LIN {X 0,Y 160.233,Z 340.194,A -85,B 0,C 180,E1 -26280.001,E2 -26280.001} C_VEL
LIN {X 0,Y 166.329,Z 331.475,A -85,B 0,C 180,E1 -26281.824,E2 -26281.824} C_VEL
LIN {X 0,Y 172.518,Z 320.915,A -85,B 0,C 180,E1 -26283.53,E2 -26283.53} C_VEL
LIN {X 0,Y 177.938,Z 309.578,A -85,B 0,C 180,E1 -26284.913,E2 -26284.913} C_VEL
LIN {X 0,Y 182.273,Z 298.101,A -85,B 0,C 180,E1 -26285.975,E2 -26285.975} C_VEL
LIN {X 0,Y 185.919,Z 285.028,A -85,B 0,C 180,E1 -26286.826,E2 -26286.826} C_VEL
LIN {X 0,Y 188.418,Z 271.569,A -85,B 0,C 180,E1 -26287.371,E2 -26287.371} C_VEL
LIN {X 0,Y 188.786,Z 268.726,A -85,B 0,C 180,E1 -26287.476,E2 -26287.476} C_VEL
LIN {X 0,Y 187.979,Z 266.198,A -85,B 0,C 180,E1 -26288.985,E2 -26288.985} C_VEL
LIN {X 0,Y 186.573,Z 263.076,A -85,B 0,C 180,E1 -26292.26,E2 -26292.26} C_VEL
LIN {X 0,Y 185.638,Z 260.546,A -85,B 0,C 180,E1 -26296.638,E2 -26296.638} C_VEL
LIN {X 0,Y 185.466,Z 260.699,A -85,B 0,C 180,E1 -26299.226,E2 -26299.226} C_VEL
LIN {X 0,Y 185.624,Z 261.538,A -85,B 0,C 180,E1 -26301.451,E2 -26301.451} C_VEL
LIN {X 0,Y 186.516,Z 265.492,A -85,B 0,C 180,E1 -26305.669,E2 -26305.669} C_VEL
LIN {X 0,Y 187.489,Z 269.73,A -85,B 0,C 180,E1 -26308.373,E2 -26308.373} C_VEL
LIN {X 0,Y 188.311,Z 273.021,A -85,B 0,C 180,E1 -26310.049,E2 -26310.049} C_VEL
LIN {X 0,Y 185.957,Z 286.979,A -85,B 0,C 180,E1 -26310.584,E2 -26310.584} C_VEL
LIN {X 0,Y 182.286,Z 300.423,A -85,B 0,C 180,E1 -26311.258,E2 -26311.258} C_VEL
LIN {X 0,Y 177.515,Z 313.155,A -85,B 0,C 180,E1 -26312.191,E2 -26312.191} C_VEL
LIN {X 0,Y 171.61,Z 325.353,A -85,B 0,C 180,E1 -26313.441,E2 -26313.441} C_VEL
LIN {X 0,Y 165.133,Z 336.315,A -85,B 0,C 180,E1 -26314.986,E2 -26314.986} C_VEL
LIN {X 0,Y 158.089,Z 346.198,A -85,B 0,C 180,E1 -26316.848,E2 -26316.848} C_VEL
LIN {X 0,Y 150.033,Z 355.815,A -85,B 0,C 180,E1 -26319.382,E2 -26319.382} C_VEL
LIN {X 0,Y 143.561,Z 362.421,A -85,B 0,C 180,E1 -26321.704,E2 -26321.704} C_VEL
LIN {X 0,Y 137.635,Z 367.953,A -85,B 0,C 180,E1 -26324.365,E2 -26324.365} C_VEL
LIN {X 0,Y 130.825,Z 373.459,A -85,B 0,C 180,E1 -26327.814,E2 -26327.814} C_VEL
LIN {X 0,Y 124.739,Z 377.873,A -85,B 0,C 180,E1 -26331.699,E2 -26331.699} C_VEL
LIN {X 0,Y 117.665,Z 382.218,A -85,B 0,C 180,E1 -26337.48,E2 -26337.48} C_VEL
LIN {X 0,Y 114.58,Z 383.794,A -85,B 0,C 180,E1 -26340.611,E2 -26340.611} C_VEL
LIN {X 0,Y 109.675,Z 385.745,A -85,B 0,C 180,E1 -26347.386,E2 -26347.386} C_VEL
LIN {X 0,Y 106.621,Z 386.253,A -85,B 0,C 180,E1 -26354.71,E2 -26354.71} C_VEL
LIN {X 0,Y 105.796,Z 385.958,A -85,B 0,C 180,E1 -26358.502,E2 -26358.502} C_VEL
LIN {X 0,Y 105.382,Z 384.173,A -85,B 0,C 180,E1 -26366.174,E2 -26366.174} C_VEL
LIN {X 0,Y 105.627,Z 382.684,A -85,B 0,C 180,E1 -26369.998,E2 -26369.998} C_VEL
LIN {X 0,Y 105.445,Z 379.479,A -85,B 0,C 180,E1 -26375.736,E2 -26375.736} C_VEL
LIN {X 0,Y 105.949,Z 375.143,A -85,B 0,C 180,E1 -26381.476,E2 -26381.476} C_VEL
LIN {X 0,Y 107.231,Z 369.534,A -85,B 0,C 180,E1 -26387.151,E2 -26387.151} C_VEL
LIN {X 0,Y 109.528,Z 362.495,A -85,B 0,C 180,E1 -26392.641,E2 -26392.641} C_VEL
LIN {X 0,Y 112.586,Z 353.593,A -85,B 0,C 180,E1 -26397.914,E2 -26397.914} C_VEL
LIN {X 0,Y 116.234,Z 343.804,A -85,B 0,C 180,E1 -26402.31,E2 -26402.31} C_VEL
LIN {X 0,Y 119.878,Z 333.229,A -85,B 0,C 180,E1 -26405.89,E2 -26405.89} C_VEL
LIN {X 0,Y 123.364,Z 321.863,A -85,B 0,C 180,E1 -26408.802,E2 -26408.802} C_VEL
LIN {X 0,Y 126.427,Z 310.142,A -85,B 0,C 180,E1 -26411.043,E2 -26411.043} C_VEL
LIN {X 0,Y 127.768,Z 304.244,A -85,B 0,C 180,E1 -26411.915,E2 -26411.915} C_VEL
LIN {X 0,Y 128.3,Z 298.694,A -85,B 0,C 180,E1 -26412.766,E2 -26412.766} C_VEL
LIN {X 0,Y 127.436,Z 289.443,A -85,B 0,C 180,E1 -26414.362,E2 -26414.362} C_VEL
LIN {X 0,Y 126.129,Z 280.088,A -85,B 0,C 180,E1 -26415.771,E2 -26415.771} C_VEL
LIN {X 0,Y 126.029,Z 274.273,A -85,B 0,C 180,E1 -26416.291,E2 -26416.291} C_VEL
LIN {X 0,Y 128.319,Z 245.916,A -85,B 0,C 180,E1 -26417.859,E2 -26417.859} C_VEL
LIN {X 0,Y 127.617,Z 235.927,A -85,B 0,C 180,E1 -26418.895,E2 -26418.895} C_VEL
LIN {X 0,Y 122.358,Z 220.14,A -85,B 0,C 180,E1 -26422.064,E2 -26422.064} C_VEL
LIN {X 0,Y 116.899,Z 206.665,A -85,B 0,C 180,E1 -26425.56,E2 -26425.56} C_VEL
LIN {X 0,Y 111.473,Z 197.493,A -85,B 0,C 180,E1 -26429.052,E2 -26429.052} C_VEL
LIN {X 0,Y 108.315,Z 192.741,A -85,B 0,C 180,E1 -26431.276,E2 -26431.276} C_VEL
LIN {X 0,Y 106.676,Z 190.164,A -85,B 0,C 180,E1 -26432.535,E2 -26432.535} C_VEL
LIN {X 0,Y 104.643,Z 187.418,A -85,B 0,C 180,E1 -26434.114,E2 -26434.114} C_VEL
LIN {X 0,Y 103.842,Z 185.904,A -85,B 0,C 180,E1 -26434.814,E2 -26434.814} C_VEL
LIN {X 0,Y 101.804,Z 183.712,A -85,B 0,C 180,E1 -26436.475,E2 -26436.475} C_VEL
LIN {X 0,Y 100.819,Z 180.918,A -85,B 0,C 180,E1 -26437.723,E2 -26437.723} C_VEL
LIN {X 0,Y 101.094,Z 180.891,A -85,B 0,C 180,E1 -26446.713,E2 -26446.713} C_VEL
LIN {X 0,Y 101.261,Z 180.849,A -85,B 0,C 180,E1 -26452.019,E2 -26452.019} C_VEL
LIN {X 0,Y 101.867,Z 180.78,A -85,B 0,C 180,E1 -26459.998,E2 -26459.998} C_VEL
LIN {X 0,Y 101.264,Z 180.871,A -85,B 0,C 180,E1 -26467.976,E2 -26467.976} C_VEL
LIN {X 0,Y 101.121,Z 180.858,A -85,B 0,C 180,E1 -26473.351,E2 -26473.351} C_VEL
LIN {X 0,Y 100.815,Z 180.924,A -85,B 0,C 180,E1 -26480.397,E2 -26480.397} C_VEL
LIN {X 0,Y 100.77,Z 180.899,A -85,B 0,C 180,E1 -26484.957,E2 -26484.957} C_VEL
LIN {X 0,Y 100.706,Z 180.927,A -85,B 0,C 180,E1 -26493.133,E2 -26493.133} C_VEL
LIN {X 0,Y 100.723,Z 180.929,A -85,B 0,C 180,E1 -26499.871,E2 -26499.871} C_VEL
LIN {X 0,Y 100.749,Z 180.912,A -85,B 0,C 180,E1 -26505.77,E2 -26505.77} C_VEL
LIN {X 0,Y 100.727,Z 180.937,A -85,B 0,C 180,E1 -26511.103,E2 -26511.103} C_VEL
LIN {X 0,Y 100.707,Z 180.933,A -85,B 0,C 180,E1 -26516.866,E2 -26516.866} C_VEL
LIN {X 0,Y 100.677,Z 180.943,A -85,B 0,C 180,E1 -26521.175,E2 -26521.175} C_VEL
LIN {X 0,Y 101.611,Z 183.625,A -85,B 0,C 180,E1 -26522.235,E2 -26522.235} C_VEL
LIN {X 0,Y 103.67,Z 185.856,A -85,B 0,C 180,E1 -26523.923,E2 -26523.923} C_VEL
LIN {X 0,Y 104.397,Z 186.604,A -85,B 0,C 180,E1 -26524.484,E2 -26524.484} C_VEL
LIN {X 0,Y 106.409,Z 189.752,A -85,B 0,C 180,E1 -26526.107,E2 -26526.107} C_VEL
LIN {X 0,Y 107.849,Z 191.69,A -85,B 0,C 180,E1 -26527.194,E2 -26527.194} C_VEL
LIN {X 0,Y 112.897,Z 199.282,A -85,B 0,C 180,E1 -26530.72,E2 -26530.72} C_VEL
LIN {X 0,Y 117.907,Z 207.42,A -85,B 0,C 180,E1 -26533.807,E2 -26533.807} C_VEL
LIN {X 0,Y 125.125,Z 221.433,A -85,B 0,C 180,E1 -26537.922,E2 -26537.922} C_VEL
LIN {X 0,Y 129.197,Z 232.015,A -85,B 0,C 180,E1 -26540.167,E2 -26540.167} C_VEL
LIN {X 0,Y 125.432,Z 274.357,A -85,B 0,C 180,E1 -26542.51,E2 -26542.51} C_VEL
LIN {X 0,Y 123.412,Z 288.198,A -85,B 0,C 180,E1 -26543.872,E2 -26543.872} C_VEL
LIN {X 0,Y 121.046,Z 300.183,A -85,B 0,C 180,E1 -26545.632,E2 -26545.632} C_VEL
LIN {X 0,Y 117.924,Z 312.467,A -85,B 0,C 180,E1 -26548.124,E2 -26548.124} C_VEL
LIN {X 0,Y 114.128,Z 324.389,A -85,B 0,C 180,E1 -26551.325,E2 -26551.325} C_VEL
LIN {X 0,Y 110.537,Z 334.612,A -85,B 0,C 180,E1 -26555.018,E2 -26555.018} C_VEL
LIN {X 0,Y 106.892,Z 344.199,A -85,B 0,C 180,E1 -26559.534,E2 -26559.534} C_VEL
LIN {X 0,Y 103.736,Z 352.637,A -85,B 0,C 180,E1 -26564.72,E2 -26564.72} C_VEL
LIN {X 0,Y 101.152,Z 359.661,A -85,B 0,C 180,E1 -26570.331,E2 -26570.331} C_VEL
LIN {X 0,Y 99.286,Z 365.396,A -85,B 0,C 180,E1 -26576.26,E2 -26576.26} C_VEL
LIN {X 0,Y 98.025,Z 370.249,A -85,B 0,C 180,E1 -26582.849,E2 -26582.849} C_VEL
LIN {X 0,Y 97.822,Z 374.211,A -85,B 0,C 180,E1 -26590.289,E2 -26590.289} C_VEL
LIN {X 0,Y 98.496,Z 376.154,A -85,B 0,C 180,E1 -26595.526,E2 -26595.526} C_VEL
LIN {X 0,Y 99.918,Z 377.48,A -85,B 0,C 180,E1 -26600.728,E2 -26600.728} C_VEL
LIN {X 0,Y 102.418,Z 378.187,A -85,B 0,C 180,E1 -26606.707,E2 -26606.707} C_VEL
LIN {X 0,Y 105.825,Z 378.009,A -85,B 0,C 180,E1 -26612.3,E2 -26612.3} C_VEL
LIN {X 0,Y 110.113,Z 376.968,A -85,B 0,C 180,E1 -26617.486,E2 -26617.486} C_VEL
LIN {X 0,Y 117.115,Z 374.207,A -85,B 0,C 180,E1 -26623.778,E2 -26623.778} C_VEL
LIN {X 0,Y 124.851,Z 370.01,A -85,B 0,C 180,E1 -26629.013,E2 -26629.013} C_VEL
LIN {X 0,Y 132.704,Z 364.735,A -85,B 0,C 180,E1 -26633.233,E2 -26633.233} C_VEL
LIN {X 0,Y 140.792,Z 358.262,A -85,B 0,C 180,E1 -26636.742,E2 -26636.742} C_VEL
LIN {X 0,Y 148.978,Z 350.375,A -85,B 0,C 180,E1 -26639.778,E2 -26639.778} C_VEL
LIN {X 0,Y 157.176,Z 341.077,A -85,B 0,C 180,E1 -26642.302,E2 -26642.302} C_VEL
LIN {X 0,Y 164.233,Z 331.414,A -85,B 0,C 180,E1 -26644.264,E2 -26644.264} C_VEL
LIN {X 0,Y 170.344,Z 321.314,A -85,B 0,C 180,E1 -26645.802,E2 -26645.802} C_VEL
LIN {X 0,Y 176.076,Z 309.663,A -85,B 0,C 180,E1 -26647.155,E2 -26647.155} C_VEL
LIN {X 0,Y 180.601,Z 297.942,A -85,B 0,C 180,E1 -26648.173,E2 -26648.173} C_VEL
LIN {X 0,Y 184.166,Z 285.441,A -85,B 0,C 180,E1 -26648.946,E2 -26648.946} C_VEL
LIN {X 0,Y 186.585,Z 273.08,A -85,B 0,C 180,E1 -26649.439,E2 -26649.439} C_VEL
LIN {X 0,Y 185.37,Z 269.984,A -85,B 0,C 180,E1 -26652.607,E2 -26652.607} C_VEL
LIN {X 0,Y 184.57,Z 267.581,A -85,B 0,C 180,E1 -26656.737,E2 -26656.737} C_VEL
LIN {X 0,Y 184.407,Z 267.621,A -85,B 0,C 180,E1 -26658.78,E2 -26658.78} C_VEL
LIN {X 0,Y 184.513,Z 268.464,A -85,B 0,C 180,E1 -26661.046,E2 -26661.046} C_VEL
LIN {X 0,Y 185.168,Z 272.044,A -85,B 0,C 180,E1 -26664.925,E2 -26664.925} C_VEL
LIN {X 0,Y 185.924,Z 276.177,A -85,B 0,C 180,E1 -26667.586,E2 -26667.586} C_VEL
LIN {X 0,Y 186.077,Z 277.273,A -85,B 0,C 180,E1 -26668.108,E2 -26668.108} C_VEL
LIN {X 0,Y 183.263,Z 290.946,A -85,B 0,C 180,E1 -26668.62,E2 -26668.62} C_VEL
LIN {X 0,Y 179.064,Z 304.295,A -85,B 0,C 180,E1 -26669.333,E2 -26669.333} C_VEL
LIN {X 0,Y 173.92,Z 316.593,A -85,B 0,C 180,E1 -26670.257,E2 -26670.257} C_VEL
LIN {X 0,Y 167.904,Z 327.975,A -85,B 0,C 180,E1 -26671.475,E2 -26671.475} C_VEL
LIN {X 0,Y 160.499,Z 339.366,A -85,B 0,C 180,E1 -26673.125,E2 -26673.125} C_VEL
LIN {X 0,Y 154.007,Z 347.754,A -85,B 0,C 180,E1 -26674.77,E2 -26674.77} C_VEL
LIN {X 0,Y 145.684,Z 356.975,A -85,B 0,C 180,E1 -26677.249,E2 -26677.249} C_VEL
LIN {X 0,Y 138.98,Z 363.363,A -85,B 0,C 180,E1 -26679.538,E2 -26679.538} C_VEL
LIN {X 0,Y 132.809,Z 368.671,A -85,B 0,C 180,E1 -26682.193,E2 -26682.193} C_VEL
LIN {X 0,Y 125.673,Z 373.97,A -85,B 0,C 180,E1 -26685.648,E2 -26685.648} C_VEL
LIN {X 0,Y 119.246,Z 378.166,A -85,B 0,C 180,E1 -26689.583,E2 -26689.583} C_VEL
LIN {X 0,Y 111.733,Z 382.295,A -85,B 0,C 180,E1 -26695.519,E2 -26695.519} C_VEL
LIN {X 0,Y 105.609,Z 384.82,A -85,B 0,C 180,E1 -26702.233,E2 -26702.233} C_VEL
LIN {X 0,Y 101.151,Z 385.886,A -85,B 0,C 180,E1 -26709.669,E2 -26709.669} C_VEL
LIN {X 0,Y 98.835,Z 385.455,A -85,B 0,C 180,E1 -26717.68,E2 -26717.68} C_VEL
LIN {X 0,Y 98.306,Z 383.517,A -85,B 0,C 180,E1 -26725.898,E2 -26725.898} C_VEL
LIN {X 0,Y 98.573,Z 381.956,A -85,B 0,C 180,E1 -26729.998,E2 -26729.998} C_VEL
LIN {X 0,Y 98.39,Z 378.59,A -85,B 0,C 180,E1 -26736.148,E2 -26736.148} C_VEL
LIN {X 0,Y 98.984,Z 374.082,A -85,B 0,C 180,E1 -26742.296,E2 -26742.296} C_VEL
LIN {X 0,Y 100.799,Z 367.149,A -85,B 0,C 180,E1 -26749.338,E2 -26749.338} C_VEL
LIN {X 0,Y 103.505,Z 359.608,A -85,B 0,C 180,E1 -26755.109,E2 -26755.109} C_VEL
LIN {X 0,Y 106.341,Z 351.85,A -85,B 0,C 180,E1 -26759.711,E2 -26759.711} C_VEL
LIN {X 0,Y 110.101,Z 342.13,A -85,B 0,C 180,E1 -26764.115,E2 -26764.115} C_VEL
LIN {X 0,Y 113.71,Z 332.002,A -85,B 0,C 180,E1 -26767.612,E2 -26767.612} C_VEL
LIN {X 0,Y 117.42,Z 320.485,A -85,B 0,C 180,E1 -26770.608,E2 -26770.608} C_VEL
LIN {X 0,Y 120.653,Z 308.395,A -85,B 0,C 180,E1 -26772.903,E2 -26772.903} C_VEL
LIN {X 0,Y 123.371,Z 295.237,A -85,B 0,C 180,E1 -26774.68,E2 -26774.68} C_VEL
LIN {X 0,Y 125.293,Z 282.442,A -85,B 0,C 180,E1 -26775.799,E2 -26775.799} C_VEL
LIN {X 0,Y 126.029,Z 274.273,A -85,B 0,C 180,E1 -26776.291,E2 -26776.291} C_VEL
LIN {X 0,Y 126.035,Z 268.462,A -85,B 0,C 180,E1 -26776.759,E2 -26776.759} C_VEL
LIN {X 0,Y 124.727,Z 259.017,A -85,B 0,C 180,E1 -26777.932,E2 -26777.932} C_VEL
LIN {X 0,Y 123.318,Z 251.52,A -85,B 0,C 180,E1 -26779.016,E2 -26779.016} C_VEL
LIN {X 0,Y 122.351,Z 243.901,A -85,B 0,C 180,E1 -26779.997,E2 -26779.997} C_VEL
LIN {X 0,Y 121.929,Z 238.108,A -85,B 0,C 180,E1 -26780.649,E2 -26780.649} C_VEL
LIN {X 0,Y 117.441,Z 224.046,A -85,B 0,C 180,E1 -26783.657,E2 -26783.657} C_VEL
LIN {X 0,Y 112.403,Z 211.152,A -85,B 0,C 180,E1 -26787.163,E2 -26787.163} C_VEL
LIN {X 0,Y 107.107,Z 201.943,A -85,B 0,C 180,E1 -26790.905,E2 -26790.905} C_VEL
LIN {X 0,Y 102.944,Z 195.483,A -85,B 0,C 180,E1 -26794.212,E2 -26794.212} C_VEL
LIN {X 0,Y 100.08,Z 191.295,A -85,B 0,C 180,E1 -26796.694,E2 -26796.694} C_VEL
LIN {X 0,Y 97.932,Z 188.228,A -85,B 0,C 180,E1 -26798.73,E2 -26798.73} C_VEL
LIN {X 0,Y 97.319,Z 187.092,A -85,B 0,C 180,E1 -26799.385,E2 -26799.385} C_VEL
LIN {X 0,Y 95.008,Z 185.052,A -85,B 0,C 180,E1 -26801.674,E2 -26801.674} C_VEL
LIN {X 0,Y 93.897,Z 182.427,A -85,B 0,C 180,E1 -26803.132,E2 -26803.132} C_VEL
LIN {X 0,Y 93.809,Z 181.783,A -85,B 0,C 180,E1 -26803.394,E2 -26803.394} C_VEL
LIN {X 0,Y 94.062,Z 181.768,A -85,B 0,C 180,E1 -26807.045,E2 -26807.045} C_VEL
LIN {X 0,Y 94.192,Z 181.73,A -85,B 0,C 180,E1 -26811.416,E2 -26811.416} C_VEL
LIN {X 0,Y 94.793,Z 181.659,A -85,B 0,C 180,E1 -26819.998,E2 -26819.998} C_VEL
LIN {X 0,Y 94.197,Z 181.751,A -85,B 0,C 180,E1 -26828.579,E2 -26828.579} C_VEL
LIN {X 0,Y 94.039,Z 181.739,A -85,B 0,C 180,E1 -26833.708,E2 -26833.708} C_VEL
LIN {X 0,Y 93.69,Z 181.802,A -85,B 0,C 180,E1 -26842.026,E2 -26842.026} C_VEL
LIN {X 0,Y 93.619,Z 181.791,A -85,B 0,C 180,E1 -26846.768,E2 -26846.768} C_VEL
LIN {X 0,Y 93.618,Z 181.799,A -85,B 0,C 180,E1 -26854.336,E2 -26854.336} C_VEL
LIN {X 0,Y 93.645,Z 181.814,A -85,B 0,C 180,E1 -26862.486,E2 -26862.486} C_VEL
LIN {X 0,Y 93.644,Z 181.808,A -85,B 0,C 180,E1 -26868.63,E2 -26868.63} C_VEL
LIN {X 0,Y 93.605,Z 181.809,A -85,B 0,C 180,E1 -26875.354,E2 -26875.354} C_VEL
LIN {X 0,Y 94.576,Z 184.497,A -85,B 0,C 180,E1 -26876.699,E2 -26876.699} C_VEL
LIN {X 0,Y 96.422,Z 186.628,A -85,B 0,C 180,E1 -26878.655,E2 -26878.655} C_VEL
LIN {X 0,Y 97.443,Z 187.526,A -85,B 0,C 180,E1 -26879.636,E2 -26879.636} C_VEL
LIN {X 0,Y 99.279,Z 190.545,A -85,B 0,C 180,E1 -26881.492,E2 -26881.492} C_VEL
LIN {X 0,Y 101.113,Z 192.633,A -85,B 0,C 180,E1 -26883.086,E2 -26883.086} C_VEL
LIN {X 0,Y 104.658,Z 197.834,A -85,B 0,C 180,E1 -26886.016,E2 -26886.016} C_VEL
LIN {X 0,Y 109.424,Z 205.272,A -85,B 0,C 180,E1 -26889.593,E2 -26889.593} C_VEL
LIN {X 0,Y 113.895,Z 212.833,A -85,B 0,C 180,E1 -26892.573,E2 -26892.573} C_VEL
LIN {X 0,Y 120.275,Z 225.658,A -85,B 0,C 180,E1 -26896.485,E2 -26896.485} C_VEL
LIN {X 0,Y 123.282,Z 234.132,A -85,B 0,C 180,E1 -26898.353,E2 -26898.353} C_VEL
LIN {X 0,Y 119.557,Z 274.458,A -85,B 0,C 180,E1 -26900.646,E2 -26900.646} C_VEL
LIN {X 0,Y 117.566,Z 287.596,A -85,B 0,C 180,E1 -26901.948,E2 -26901.948} C_VEL
LIN {X 0,Y 115.013,Z 300.17,A -85,B 0,C 180,E1 -26903.82,E2 -26903.82} C_VEL
LIN {X 0,Y 111.733,Z 312.533,A -85,B 0,C 180,E1 -26906.396,E2 -26906.396} C_VEL
LIN {X 0,Y 107.971,Z 323.898,A -85,B 0,C 180,E1 -26909.536,E2 -26909.536} C_VEL
LIN {X 0,Y 104.172,Z 334.203,A -85,B 0,C 180,E1 -26913.328,E2 -26913.328} C_VEL
LIN {X 0,Y 100.316,Z 343.88,A -85,B 0,C 180,E1 -26918.057,E2 -26918.057} C_VEL
LIN {X 0,Y 96.901,Z 352.544,A -85,B 0,C 180,E1 -26923.636,E2 -26923.636} C_VEL
LIN {X 0,Y 94.146,Z 359.676,A -85,B 0,C 180,E1 -26929.631,E2 -26929.631} C_VEL
LIN {X 0,Y 92.247,Z 365.25,A -85,B 0,C 180,E1 -26935.712,E2 -26935.712} C_VEL
LIN {X 0,Y 90.942,Z 370.167,A -85,B 0,C 180,E1 -26942.752,E2 -26942.752} C_VEL
LIN {X 0,Y 90.663,Z 373.561,A -85,B 0,C 180,E1 -26949.183,E2 -26949.183} C_VEL
LIN {X 0,Y 91.501,Z 376.25,A -85,B 0,C 180,E1 -26956.272,E2 -26956.272} C_VEL
LIN {X 0,Y 93.466,Z 377.886,A -85,B 0,C 180,E1 -26963.022,E2 -26963.022} C_VEL
LIN {X 0,Y 97.027,Z 378.582,A -85,B 0,C 180,E1 -26970.371,E2 -26970.371} C_VEL
LIN {X 0,Y 100.488,Z 378.319,A -85,B 0,C 180,E1 -26975.402,E2 -26975.402} C_VEL
LIN {X 0,Y 105.082,Z 377.273,A -85,B 0,C 180,E1 -26980.466,E2 -26980.466} C_VEL
LIN {X 0,Y 110.669,Z 375.334,A -85,B 0,C 180,E1 -26985.287,E2 -26985.287} C_VEL
LIN {X 0,Y 118.62,Z 371.612,A -85,B 0,C 180,E1 -26990.613,E2 -26990.613} C_VEL
LIN {X 0,Y 126.986,Z 366.619,A -85,B 0,C 180,E1 -26995.028,E2 -26995.028} C_VEL
LIN {X 0,Y 136.401,Z 359.72,A -85,B 0,C 180,E1 -26998.966,E2 -26998.966} C_VEL
LIN {X 0,Y 144.141,Z 352.917,A -85,B 0,C 180,E1 -27001.695,E2 -27001.695} C_VEL
LIN {X 0,Y 152.381,Z 344.374,A -85,B 0,C 180,E1 -27004.134,E2 -27004.134} C_VEL
LIN {X 0,Y 159.988,Z 334.827,A -85,B 0,C 180,E1 -27006.145,E2 -27006.145} C_VEL
LIN {X 0,Y 167.299,Z 323.756,A -85,B 0,C 180,E1 -27007.875,E2 -27007.875} C_VEL
LIN {X 0,Y 173.592,Z 311.856,A -85,B 0,C 180,E1 -27009.254,E2 -27009.254} C_VEL
LIN {X 0,Y 178.572,Z 299.834,A -85,B 0,C 180,E1 -27010.283,E2 -27010.283} C_VEL
LIN {X 0,Y 182.504,Z 287.095,A -85,B 0,C 180,E1 -27011.064,E2 -27011.064} C_VEL
LIN {X 0,Y 184.447,Z 278.319,A -85,B 0,C 180,E1 -27011.452,E2 -27011.452} C_VEL
LIN {X 0,Y 183.966,Z 276.707,A -85,B 0,C 180,E1 -27013.252,E2 -27013.252} C_VEL
LIN {X 0,Y 183.408,Z 274.517,A -85,B 0,C 180,E1 -27017.349,E2 -27017.349} C_VEL
LIN {X 0,Y 183.365,Z 275.226,A -85,B 0,C 180,E1 -27020.466,E2 -27020.466} C_VEL
LIN {X 0,Y 183.767,Z 278.831,A -85,B 0,C 180,E1 -27024.334,E2 -27024.334} C_VEL
LIN {X 0,Y 184.052,Z 281.28,A -85,B 0,C 180,E1 -27026.017,E2 -27026.017} C_VEL
LIN {X 0,Y 180.937,Z 294.125,A -85,B 0,C 180,E1 -27026.571,E2 -27026.571} C_VEL
LIN {X 0,Y 176.384,Z 307.158,A -85,B 0,C 180,E1 -27027.274,E2 -27027.274} C_VEL
LIN {X 0,Y 170.542,Z 319.74,A -85,B 0,C 180,E1 -27028.251,E2 -27028.251} C_VEL
LIN {X 0,Y 163.604,Z 331.66,A -85,B 0,C 180,E1 -27029.552,E2 -27029.552} C_VEL
LIN {X 0,Y 156.042,Z 342.234,A -85,B 0,C 180,E1 -27031.155,E2 -27031.155} C_VEL
LIN {X 0,Y 148.685,Z 350.91,A -85,B 0,C 180,E1 -27032.962,E2 -27032.962} C_VEL
LIN {X 0,Y 140.143,Z 359.482,A -85,B 0,C 180,E1 -27035.418,E2 -27035.418} C_VEL
LIN {X 0,Y 133.38,Z 365.329,A -85,B 0,C 180,E1 -27037.777,E2 -27037.777} C_VEL
LIN {X 0,Y 125.63,Z 371.178,A -85,B 0,C 180,E1 -27040.953,E2 -27040.953} C_VEL
LIN {X 0,Y 118.362,Z 375.9,A -85,B 0,C 180,E1 -27044.556,E2 -27044.556} C_VEL
LIN {X 0,Y 111.826,Z 379.58,A -85,B 0,C 180,E1 -27048.705,E2 -27048.705} C_VEL
LIN {X 0,Y 105.949,Z 382.339,A -85,B 0,C 180,E1 -27053.342,E2 -27053.342} C_VEL
LIN {X 0,Y 99.35,Z 384.688,A -85,B 0,C 180,E1 -27060.316,E2 -27060.316} C_VEL
LIN {X 0,Y 94.499,Z 385.54,A -85,B 0,C 180,E1 -27068.167,E2 -27068.167} C_VEL
LIN {X 0,Y 91.905,Z 384.931,A -85,B 0,C 180,E1 -27076.735,E2 -27076.735} C_VEL
LIN {X 0,Y 91.255,Z 382.854,A -85,B 0,C 180,E1 -27085.58,E2 -27085.58} C_VEL
LIN {X 0,Y 91.498,Z 381.166,A -85,B 0,C 180,E1 -27089.997,E2 -27089.997} C_VEL
LIN {X 0,Y 91.36,Z 377.649,A -85,B 0,C 180,E1 -27096.624,E2 -27096.624} C_VEL
LIN {X 0,Y 92.028,Z 372.948,A -85,B 0,C 180,E1 -27103.242,E2 -27103.242} C_VEL
LIN {X 0,Y 93.705,Z 366.932,A -85,B 0,C 180,E1 -27109.722,E2 -27109.722} C_VEL
LIN {X 0,Y 96.535,Z 359.419,A -85,B 0,C 180,E1 -27115.898,E2 -27115.898} C_VEL
LIN {X 0,Y 99.513,Z 351.69,A -85,B 0,C 180,E1 -27120.796,E2 -27120.796} C_VEL
LIN {X 0,Y 103.226,Z 342.6,A -85,B 0,C 180,E1 -27125.21,E2 -27125.21} C_VEL
LIN {X 0,Y 107.237,Z 331.939,A -85,B 0,C 180,E1 -27129.106,E2 -27129.106} C_VEL
LIN {X 0,Y 111.095,Z 320.47,A -85,B 0,C 180,E1 -27132.231,E2 -27132.231} C_VEL
LIN {X 0,Y 114.459,Z 308.497,A -85,B 0,C 180,E1 -27134.608,E2 -27134.608} C_VEL
LIN {X 0,Y 117.417,Z 294.939,A -85,B 0,C 180,E1 -27136.495,E2 -27136.495} C_VEL
LIN {X 0,Y 119.428,Z 281.907,A -85,B 0,C 180,E1 -27137.665,E2 -27137.665} C_VEL
LIN {X 0,Y 122.51,Z 246.783,A -85,B 0,C 180,E1 -27139.693,E2 -27139.693} C_VEL
LIN {X 0,Y 122.351,Z 243.901,A -85,B 0,C 180,E1 -27139.997,E2 -27139.997} C_VEL
LIN {X 0,Y 121.71,Z 240.236,A -85,B 0,C 180,E1 -27140.543,E2 -27140.543} C_VEL
LIN {X 0,Y 120.468,Z 236.88,A -85,B 0,C 180,E1 -27141.295,E2 -27141.295} C_VEL
LIN {X 0,Y 116.944,Z 230.966,A -85,B 0,C 180,E1 -27143.21,E2 -27143.21} C_VEL
LIN {X 0,Y 111.045,Z 222.501,A -85,B 0,C 180,E1 -27146.641,E2 -27146.641} C_VEL
LIN {X 0,Y 109.458,Z 219.349,A -85,B 0,C 180,E1 -27147.733,E2 -27147.733} C_VEL
LIN {X 0,Y 107.063,Z 213.848,A -85,B 0,C 180,E1 -27149.574,E2 -27149.574} C_VEL
LIN {X 0,Y 101.847,Z 204.644,A -85,B 0,C 180,E1 -27153.77,E2 -27153.77} C_VEL
LIN {X 0,Y 98.777,Z 200.068,A -85,B 0,C 180,E1 -27156.435,E2 -27156.435} C_VEL
LIN {X 0,Y 96.5,Z 196.602,A -85,B 0,C 180,E1 -27158.643,E2 -27158.643} C_VEL
LIN {X 0,Y 94.108,Z 193.001,A -85,B 0,C 180,E1 -27161.21,E2 -27161.21} C_VEL
LIN {X 0,Y 91.854,Z 190.437,A -85,B 0,C 180,E1 -27163.752,E2 -27163.752} C_VEL
LIN {X 0,Y 90.636,Z 188.067,A -85,B 0,C 180,E1 -27165.401,E2 -27165.401} C_VEL
LIN {X 0,Y 88.164,Z 185.728,A -85,B 0,C 180,E1 -27168.648,E2 -27168.648} C_VEL
LIN {X 0,Y 87.181,Z 183.289,A -85,B 0,C 180,E1 -27170.427,E2 -27170.427} C_VEL
LIN {X 0,Y 87.107,Z 182.614,A -85,B 0,C 180,E1 -27170.858,E2 -27170.858} C_VEL
LIN {X 0,Y 87.72,Z 182.539,A -85,B 0,C 180,E1 -27179.997,E2 -27179.997} C_VEL
LIN {X 0,Y 87.105,Z 182.631,A -85,B 0,C 180,E1 -27189.284,E2 -27189.284} C_VEL
LIN {X 0,Y 86.946,Z 182.622,A -85,B 0,C 180,E1 -27194.085,E2 -27194.085} C_VEL
LIN {X 0,Y 86.66,Z 182.687,A -85,B 0,C 180,E1 -27198.926,E2 -27198.926} C_VEL
LIN {X 0,Y 86.581,Z 182.667,A -85,B 0,C 180,E1 -27206.766,E2 -27206.766} C_VEL
LIN {X 0,Y 86.546,Z 182.672,A -85,B 0,C 180,E1 -27215.707,E2 -27215.707} C_VEL
LIN {X 0,Y 86.569,Z 182.69,A -85,B 0,C 180,E1 -27223.063,E2 -27223.063} C_VEL
LIN {X 0,Y 86.63,Z 182.783,A -85,B 0,C 180,E1 -27227.559,E2 -27227.559} C_VEL
LIN {X 0,Y 87.432,Z 185.323,A -85,B 0,C 180,E1 -27229.204,E2 -27229.204} C_VEL
LIN {X 0,Y 89.292,Z 187.497,A -85,B 0,C 180,E1 -27231.909,E2 -27231.909} C_VEL
LIN {X 0,Y 90.834,Z 188.586,A -85,B 0,C 180,E1 -27233.786,E2 -27233.786} C_VEL
LIN {X 0,Y 92.752,Z 191.879,A -85,B 0,C 180,E1 -27236.231,E2 -27236.231} C_VEL
LIN {X 0,Y 94.494,Z 193.623,A -85,B 0,C 180,E1 -27238.077,E2 -27238.077} C_VEL
LIN {X 0,Y 96.836,Z 197.115,A -85,B 0,C 180,E1 -27240.56,E2 -27240.56} C_VEL
LIN {X 0,Y 98.225,Z 199.073,A -85,B 0,C 180,E1 -27241.898,E2 -27241.898} C_VEL
LIN {X 0,Y 101.072,Z 203.296,A -85,B 0,C 180,E1 -27244.444,E2 -27244.444} C_VEL
LIN {X 0,Y 107.252,Z 213.206,A -85,B 0,C 180,E1 -27249.314,E2 -27249.314} C_VEL
LIN {X 0,Y 112.021,Z 222.621,A -85,B 0,C 180,E1 -27252.7,E2 -27252.7} C_VEL
LIN {X 0,Y 115.461,Z 229.809,A -85,B 0,C 180,E1 -27254.908,E2 -27254.908} C_VEL
LIN {X 0,Y 117.569,Z 235.73,A -85,B 0,C 180,E1 -27256.337,E2 -27256.337} C_VEL
LIN {X 0,Y 113.833,Z 274.465,A -85,B 0,C 180,E1 -27258.583,E2 -27258.583} C_VEL
LIN {X 0,Y 111.733,Z 287.778,A -85,B 0,C 180,E1 -27259.927,E2 -27259.927} C_VEL
LIN {X 0,Y 109.004,Z 300.609,A -85,B 0,C 180,E1 -27261.894,E2 -27261.894} C_VEL
LIN {X 0,Y 105.678,Z 312.537,A -85,B 0,C 180,E1 -27264.452,E2 -27264.452} C_VEL
LIN {X 0,Y 101.928,Z 323.393,A -85,B 0,C 180,E1 -27267.532,E2 -27267.532} C_VEL
LIN {X 0,Y 97.941,Z 333.704,A -85,B 0,C 180,E1 -27271.425,E2 -27271.425} C_VEL
LIN {X 0,Y 93.759,Z 343.649,A -85,B 0,C 180,E1 -27276.458,E2 -27276.458} C_VEL
LIN {X 0,Y 90.101,Z 352.388,A -85,B 0,C 180,E1 -27282.389,E2 -27282.389} C_VEL
LIN {X 0,Y 87.176,Z 359.594,A -85,B 0,C 180,E1 -27288.815,E2 -27288.815} C_VEL
LIN {X 0,Y 85.256,Z 364.899,A -85,B 0,C 180,E1 -27294.944,E2 -27294.944} C_VEL
LIN {X 0,Y 83.803,Z 370.256,A -85,B 0,C 180,E1 -27303.009,E2 -27303.009} C_VEL
LIN {X 0,Y 83.768,Z 374.566,A -85,B 0,C 180,E1 -27312.163,E2 -27312.163} C_VEL
LIN {X 0,Y 84.821,Z 376.692,A -85,B 0,C 180,E1 -27318.486,E2 -27318.486} C_VEL
LIN {X 0,Y 87.186,Z 378.281,A -85,B 0,C 180,E1 -27325.652,E2 -27325.652} C_VEL
LIN {X 0,Y 90.621,Z 378.929,A -85,B 0,C 180,E1 -27332.272,E2 -27332.272} C_VEL
LIN {X 0,Y 96.973,Z 378.366,A -85,B 0,C 180,E1 -27340.425,E2 -27340.425} C_VEL
LIN {X 0,Y 101.852,Z 377.194,A -85,B 0,C 180,E1 -27345.032,E2 -27345.032} C_VEL
LIN {X 0,Y 110.274,Z 374.09,A -85,B 0,C 180,E1 -27351.074,E2 -27351.074} C_VEL
LIN {X 0,Y 119.739,Z 369.398,A -85,B 0,C 180,E1 -27356.229,E2 -27356.229} C_VEL
LIN {X 0,Y 128.707,Z 363.752,A -85,B 0,C 180,E1 -27360.002,E2 -27360.002} C_VEL
LIN {X 0,Y 136.958,Z 357.466,A -85,B 0,C 180,E1 -27362.943,E2 -27362.943} C_VEL
LIN {X 0,Y 145.64,Z 349.596,A -85,B 0,C 180,E1 -27365.54,E2 -27365.54} C_VEL
LIN {X 0,Y 153.843,Z 340.752,A -85,B 0,C 180,E1 -27367.628,E2 -27367.628} C_VEL
LIN {X 0,Y 161.133,Z 331.247,A -85,B 0,C 180,E1 -27369.305,E2 -27369.305} C_VEL
LIN {X 0,Y 168.118,Z 320.188,A -85,B 0,C 180,E1 -27370.759,E2 -27370.759} C_VEL
LIN {X 0,Y 173.05,Z 310.61,A -85,B 0,C 180,E1 -27371.717,E2 -27371.717} C_VEL
LIN {X 0,Y 178.017,Z 298.517,A -85,B 0,C 180,E1 -27372.648,E2 -27372.648} C_VEL
LIN {X 0,Y 181.661,Z 286.463,A -85,B 0,C 180,E1 -27373.314,E2 -27373.314} C_VEL
LIN {X 0,Y 182.368,Z 283.593,A -85,B 0,C 180,E1 -27373.441,E2 -27373.441} C_VEL
LIN {X 0,Y 182.04,Z 281.453,A -85,B 0,C 180,E1 -27377.483,E2 -27377.483} C_VEL
LIN {X 0,Y 181.958,Z 282.19,A -85,B 0,C 180,E1 -27380.18,E2 -27380.18} C_VEL
LIN {X 0,Y 182.026,Z 285.356,A -85,B 0,C 180,E1 -27383.633,E2 -27383.633} C_VEL
LIN {X 0,Y 181.981,Z 286.157,A -85,B 0,C 180,E1 -27384.04,E2 -27384.04} C_VEL
LIN {X 0,Y 177.8,Z 300.258,A -85,B 0,C 180,E1 -27384.611,E2 -27384.611} C_VEL
LIN {X 0,Y 172.667,Z 312.695,A -85,B 0,C 180,E1 -27385.339,E2 -27385.339} C_VEL
LIN {X 0,Y 166.581,Z 324.252,A -85,B 0,C 180,E1 -27386.291,E2 -27386.291} C_VEL
LIN {X 0,Y 159.525,Z 335.164,A -85,B 0,C 180,E1 -27387.545,E2 -27387.545} C_VEL
LIN {X 0,Y 151.025,Z 345.842,A -85,B 0,C 180,E1 -27389.242,E2 -27389.242} C_VEL
LIN {X 0,Y 142.041,Z 355.276,A -85,B 0,C 180,E1 -27391.401,E2 -27391.401} C_VEL
LIN {X 0,Y 133.309,Z 362.957,A -85,B 0,C 180,E1 -27393.864,E2 -27393.864} C_VEL
LIN {X 0,Y 126.48,Z 368.203,A -85,B 0,C 180,E1 -27396.318,E2 -27396.318} C_VEL
LIN {X 0,Y 118.5,Z 373.429,A -85,B 0,C 180,E1 -27399.553,E2 -27399.553} C_VEL
LIN {X 0,Y 111.129,Z 377.563,A -85,B 0,C 180,E1 -27403.338,E2 -27403.338} C_VEL
LIN {X 0,Y 103.95,Z 380.96,A -85,B 0,C 180,E1 -27408.051,E2 -27408.051} C_VEL
LIN {X 0,Y 96.565,Z 383.66,A -85,B 0,C 180,E1 -27414.389,E2 -27414.389} C_VEL
LIN {X 0,Y 90.328,Z 385.026,A -85,B 0,C 180,E1 -27422.168,E2 -27422.168} C_VEL
LIN {X 0,Y 86.166,Z 384.967,A -85,B 0,C 180,E1 -27430.955,E2 -27430.955} C_VEL
LIN {X 0,Y 84.319,Z 383.454,A -85,B 0,C 180,E1 -27440.401,E2 -27440.401} C_VEL
LIN {X 0,Y 84.371,Z 380.975,A -85,B 0,C 180,E1 -27448.439,E2 -27448.439} C_VEL
LIN {X 0,Y 84.371,Z 379.654,A -85,B 0,C 180,E1 -27451.55,E2 -27451.55} C_VEL
LIN {X 0,Y 84.489,Z 375.177,A -85,B 0,C 180,E1 -27459.574,E2 -27459.574} C_VEL
LIN {X 0,Y 85.931,Z 368.855,A -85,B 0,C 180,E1 -27467.858,E2 -27467.858} C_VEL
LIN {X 0,Y 88.485,Z 361.935,A -85,B 0,C 180,E1 -27474.641,E2 -27474.641} C_VEL
LIN {X 0,Y 91.358,Z 354.799,A -85,B 0,C 180,E1 -27479.999,E2 -27479.999} C_VEL
LIN {X 0,Y 95.074,Z 346.184,A -85,B 0,C 180,E1 -27484.949,E2 -27484.949} C_VEL
LIN {X 0,Y 99.481,Z 335.588,A -85,B 0,C 180,E1 -27489.478,E2 -27489.478} C_VEL
LIN {X 0,Y 103.316,Z 325.068,A -85,B 0,C 180,E1 -27492.859,E2 -27492.859} C_VEL
LIN {X 0,Y 106.997,Z 313.524,A -85,B 0,C 180,E1 -27495.584,E2 -27495.584} C_VEL
LIN {X 0,Y 110.346,Z 300.509,A -85,B 0,C 180,E1 -27497.763,E2 -27497.763} C_VEL
LIN {X 0,Y 112.89,Z 287.206,A -85,B 0,C 180,E1 -27499.259,E2 -27499.259} C_VEL
LIN {X 0,Y 114.63,Z 271.795,A -85,B 0,C 180,E1 -27500.312,E2 -27500.312} C_VEL
LIN {X 0,Y 116.828,Z 246.797,A -85,B 0,C 180,E1 -27501.78,E2 -27501.78} C_VEL
LIN {X 0,Y 116.412,Z 240.265,A -85,B 0,C 180,E1 -27502.555,E2 -27502.555} C_VEL
LIN {X 0,Y 112.025,Z 226.294,A -85,B 0,C 180,E1 -27505.8,E2 -27505.8} C_VEL
LIN {X 0,Y 109.458,Z 219.349,A -85,B 0,C 180,E1 -27507.733,E2 -27507.733} C_VEL
LIN {X 0,Y 107.022,Z 215.1,A -85,B 0,C 180,E1 -27509.464,E2 -27509.464} C_VEL
LIN {X 0,Y 104.026,Z 211.727,A -85,B 0,C 180,E1 -27511.559,E2 -27511.559} C_VEL
LIN {X 0,Y 93.599,Z 202.612,A -85,B 0,C 180,E1 -27520.135,E2 -27520.135} C_VEL
LIN {X 0,Y 91.05,Z 198.848,A -85,B 0,C 180,E1 -27523.1,E2 -27523.1} C_VEL
LIN {X 0,Y 88.584,Z 195.488,A -85,B 0,C 180,E1 -27526.228,E2 -27526.228} C_VEL
LIN {X 0,Y 87.886,Z 194.192,A -85,B 0,C 180,E1 -27527.27,E2 -27527.27} C_VEL
LIN {X 0,Y 85.437,Z 191.268,A -85,B 0,C 180,E1 -27531.012,E2 -27531.012} C_VEL
LIN {X 0,Y 84.663,Z 189.302,A -85,B 0,C 180,E1 -27532.605,E2 -27532.605} C_VEL
LIN {X 0,Y 82.175,Z 187.433,A -85,B 0,C 180,E1 -27537.24,E2 -27537.24} C_VEL
LIN {X 0,Y 80.31,Z 183.452,A -85,B 0,C 180,E1 -27542.819,E2 -27542.819} C_VEL
LIN {X 0,Y 79.99,Z 183.508,A -85,B 0,C 180,E1 -27550.118,E2 -27550.118} C_VEL
LIN {X 0,Y 79.762,Z 183.519,A -85,B 0,C 180,E1 -27555.325,E2 -27555.325} C_VEL
LIN {X 0,Y 79.519,Z 183.575,A -85,B 0,C 180,E1 -27560.7,E2 -27560.7} C_VEL
LIN {X 0,Y 79.48,Z 183.556,A -85,B 0,C 180,E1 -27567.847,E2 -27567.847} C_VEL
LIN {X 0,Y 79.498,Z 183.692,A -85,B 0,C 180,E1 -27573.918,E2 -27573.918} C_VEL
LIN {X 0,Y 80.58,Z 186.632,A -85,B 0,C 180,E1 -27578.045,E2 -27578.045} C_VEL
LIN {X 0,Y 83.667,Z 189.183,A -85,B 0,C 180,E1 -27584.704,E2 -27584.704} C_VEL
LIN {X 0,Y 84.374,Z 189.721,A -85,B 0,C 180,E1 -27585.921,E2 -27585.921} C_VEL
LIN {X 0,Y 85.823,Z 192.606,A -85,B 0,C 180,E1 -27588.673,E2 -27588.673} C_VEL
LIN {X 0,Y 88.241,Z 194.979,A -85,B 0,C 180,E1 -27592.169,E2 -27592.169} C_VEL
LIN {X 0,Y 90.598,Z 198.538,A -85,B 0,C 180,E1 -27595.307,E2 -27595.307} C_VEL
LIN {X 0,Y 91.783,Z 200.057,A -85,B 0,C 180,E1 -27596.687,E2 -27596.687} C_VEL
LIN {X 0,Y 95.205,Z 205.053,A -85,B 0,C 180,E1 -27600.43,E2 -27600.43} C_VEL
LIN {X 0,Y 99.259,Z 211.459,A -85,B 0,C 180,E1 -27604.298,E2 -27604.298} C_VEL
LIN {X 0,Y 104.406,Z 220.417,A -85,B 0,C 180,E1 -27608.556,E2 -27608.556} C_VEL
LIN {X 0,Y 110.509,Z 233.459,A -85,B 0,C 180,E1 -27613.109,E2 -27613.109} C_VEL
LIN {X 0,Y 111.915,Z 237.552,A -85,B 0,C 180,E1 -27614.153,E2 -27614.153} C_VEL
LIN {X 0,Y 108.275,Z 274.095,A -85,B 0,C 180,E1 -27616.321,E2 -27616.321} C_VEL
LIN {X 0,Y 106.052,Z 287.64,A -85,B 0,C 180,E1 -27617.691,E2 -27617.691} C_VEL
LIN {X 0,Y 103.187,Z 300.541,A -85,B 0,C 180,E1 -27619.703,E2 -27619.703} C_VEL
LIN {X 0,Y 99.55,Z 312.886,A -85,B 0,C 180,E1 -27622.417,E2 -27622.417} C_VEL
LIN {X 0,Y 95.416,Z 324.214,A -85,B 0,C 180,E1 -27625.778,E2 -27625.778} C_VEL
LIN {X 0,Y 91.134,Z 334.708,A -85,B 0,C 180,E1 -27630.003,E2 -27630.003} C_VEL
LIN {X 0,Y 87.286,Z 343.343,A -85,B 0,C 180,E1 -27634.621,E2 -27634.621} C_VEL
LIN {X 0,Y 83.379,Z 352.181,A -85,B 0,C 180,E1 -27640.935,E2 -27640.935} C_VEL
LIN {X 0,Y 79.983,Z 360.091,A -85,B 0,C 180,E1 -27648.503,E2 -27648.503} C_VEL
LIN {X 0,Y 77.631,Z 366.535,A -85,B 0,C 180,E1 -27656.917,E2 -27656.917} C_VEL
LIN {X 0,Y 76.574,Z 370.833,A -85,B 0,C 180,E1 -27664.312,E2 -27664.312} C_VEL
LIN {X 0,Y 76.72,Z 374.556,A -85,B 0,C 180,E1 -27672.879,E2 -27672.879} C_VEL
LIN {X 0,Y 78.954,Z 377.638,A -85,B 0,C 180,E1 -27683.243,E2 -27683.243} C_VEL
LIN {X 0,Y 81.538,Z 378.768,A -85,B 0,C 180,E1 -27689.54,E2 -27689.54} C_VEL
LIN {X 0,Y 85.083,Z 379.295,A -85,B 0,C 180,E1 -27695.609,E2 -27695.609} C_VEL
LIN {X 0,Y 90.102,Z 379.03,A -85,B 0,C 180,E1 -27701.823,E2 -27701.823} C_VEL
LIN {X 0,Y 96.005,Z 377.913,A -85,B 0,C 180,E1 -27707.316,E2 -27707.316} C_VEL
LIN {X 0,Y 102.728,Z 375.916,A -85,B 0,C 180,E1 -27712.138,E2 -27712.138} C_VEL
LIN {X 0,Y 112.552,Z 371.873,A -85,B 0,C 180,E1 -27717.581,E2 -27717.581} C_VEL
LIN {X 0,Y 121.202,Z 367.225,A -85,B 0,C 180,E1 -27721.292,E2 -27721.292} C_VEL
LIN {X 0,Y 130.433,Z 361.143,A -85,B 0,C 180,E1 -27724.547,E2 -27724.547} C_VEL
LIN {X 0,Y 139.987,Z 353.518,A -85,B 0,C 180,E1 -27727.359,E2 -27727.359} C_VEL
LIN {X 0,Y 148.137,Z 345.728,A -85,B 0,C 180,E1 -27729.327,E2 -27729.327} C_VEL
LIN {X 0,Y 156.461,Z 336.098,A -85,B 0,C 180,E1 -27731.15,E2 -27731.15} C_VEL
LIN {X 0,Y 163.768,Z 325.825,A -85,B 0,C 180,E1 -27732.582,E2 -27732.582} C_VEL
LIN {X 0,Y 170.581,Z 314.083,A -85,B 0,C 180,E1 -27733.802,E2 -27733.802} C_VEL
LIN {X 0,Y 175.775,Z 302.617,A -85,B 0,C 180,E1 -27734.705,E2 -27734.705} C_VEL
LIN {X 0,Y 180.249,Z 289.537,A -85,B 0,C 180,E1 -27735.433,E2 -27735.433} C_VEL
LIN {X 0,Y 180.313,Z 288.432,A -85,B 0,C 180,E1 -27737.331,E2 -27737.331} C_VEL
LIN {X 0,Y 180.211,Z 288.918,A -85,B 0,C 180,E1 -27739.685,E2 -27739.685} C_VEL
LIN {X 0,Y 180.013,Z 290.91,A -85,B 0,C 180,E1 -27741.963,E2 -27741.963} C_VEL
LIN {X 0,Y 175.622,Z 303.703,A -85,B 0,C 180,E1 -27742.489,E2 -27742.489} C_VEL
LIN {X 0,Y 170.128,Z 315.804,A -85,B 0,C 180,E1 -27743.197,E2 -27743.197} C_VEL
LIN {X 0,Y 163.629,Z 327.09,A -85,B 0,C 180,E1 -27744.114,E2 -27744.114} C_VEL
LIN {X 0,Y 155.635,Z 338.403,A -85,B 0,C 180,E1 -27745.422,E2 -27745.422} C_VEL
LIN {X 0,Y 147.743,Z 347.618,A -85,B 0,C 180,E1 -27746.881,E2 -27746.881} C_VEL
LIN {X 0,Y 138.521,Z 356.585,A -85,B 0,C 180,E1 -27748.928,E2 -27748.928} C_VEL
LIN {X 0,Y 128.052,Z 365.006,A -85,B 0,C 180,E1 -27751.708,E2 -27751.708} C_VEL
LIN {X 0,Y 119.621,Z 370.749,A -85,B 0,C 180,E1 -27754.658,E2 -27754.658} C_VEL
LIN {X 0,Y 111.485,Z 375.386,A -85,B 0,C 180,E1 -27757.997,E2 -27757.997} C_VEL
LIN {X 0,Y 103.949,Z 378.997,A -85,B 0,C 180,E1 -27761.948,E2 -27761.948} C_VEL
LIN {X 0,Y 94.902,Z 382.424,A -85,B 0,C 180,E1 -27768.199,E2 -27768.199} C_VEL
LIN {X 0,Y 87.244,Z 384.324,A -85,B 0,C 180,E1 -27775.671,E2 -27775.671} C_VEL
LIN {X 0,Y 81.44,Z 384.8,A -85,B 0,C 180,E1 -27784.435,E2 -27784.435} C_VEL
LIN {X 0,Y 78.101,Z 383.82,A -85,B 0,C 180,E1 -27794.335,E2 -27794.335} C_VEL
LIN {X 0,Y 77.15,Z 381.334,A -85,B 0,C 180,E1 -27804.77,E2 -27804.77} C_VEL
LIN {X 0,Y 77.4,Z 379.483,A -85,B 0,C 180,E1 -27809.997,E2 -27809.997} C_VEL
LIN {X 0,Y 77.3,Z 375.623,A -85,B 0,C 180,E1 -27817.835,E2 -27817.835} C_VEL
LIN {X 0,Y 78.528,Z 369.565,A -85,B 0,C 180,E1 -27826.907,E2 -27826.907} C_VEL
LIN {X 0,Y 80.991,Z 362.882,A -85,B 0,C 180,E1 -27834.339,E2 -27834.339} C_VEL
LIN {X 0,Y 84.557,Z 354.525,A -85,B 0,C 180,E1 -27841.294,E2 -27841.294} C_VEL
LIN {X 0,Y 88.47,Z 345.943,A -85,B 0,C 180,E1 -27846.566,E2 -27846.566} C_VEL
LIN {X 0,Y 93.111,Z 335.346,A -85,B 0,C 180,E1 -27851.355,E2 -27851.355} C_VEL
LIN {X 0,Y 97.148,Z 324.925,A -85,B 0,C 180,E1 -27854.854,E2 -27854.854} C_VEL
LIN {X 0,Y 101,Z 313.471,A -85,B 0,C 180,E1 -27857.671,E2 -27857.671} C_VEL
LIN {X 0,Y 104.505,Z 300.577,A -85,B 0,C 180,E1 -27859.901,E2 -27859.901} C_VEL
LIN {X 0,Y 107.067,Z 287.939,A -85,B 0,C 180,E1 -27861.399,E2 -27861.399} C_VEL
LIN {X 0,Y 108.699,Z 275.448,A -85,B 0,C 180,E1 -27862.326,E2 -27862.326} C_VEL
LIN {X 0,Y 111.316,Z 248.04,A -85,B 0,C 180,E1 -27863.942,E2 -27863.942} C_VEL
LIN {X 0,Y 111.048,Z 242.742,A -85,B 0,C 180,E1 -27864.584,E2 -27864.584} C_VEL
LIN {X 0,Y 107.15,Z 229.813,A -85,B 0,C 180,E1 -27867.764,E2 -27867.764} C_VEL
LIN {X 0,Y 103.3,Z 219.28,A -85,B 0,C 180,E1 -27871.069,E2 -27871.069} C_VEL
LIN {X 0,Y 98.182,Z 209.936,A -85,B 0,C 180,E1 -27875.515,E2 -27875.515} C_VEL
LIN {X 0,Y 93.599,Z 202.612,A -85,B 0,C 180,E1 -27880.135,E2 -27880.135} C_VEL
LIN {X 0,Y 90.917,Z 200.122,A -85,B 0,C 180,E1 -27883.01,E2 -27883.01} C_VEL
LIN {X 0,Y 86.32,Z 197.732,A -85,B 0,C 180,E1 -27888.465,E2 -27888.465} C_VEL
LIN {X 0,Y 81.675,Z 195.369,A -85,B 0,C 180,E1 -27895.864,E2 -27895.864} C_VEL
LIN {X 0,Y 80.504,Z 194.146,A -85,B 0,C 180,E1 -27898.423,E2 -27898.423} C_VEL
LIN {X 0,Y 78.823,Z 190.504,A -85,B 0,C 180,E1 -27903.831,E2 -27903.831} C_VEL
LIN {X 0,Y 76.387,Z 189.79,A -85,B 0,C 180,E1 -27916.019,E2 -27916.019} C_VEL
LIN {X 0,Y 77.978,Z 190.513,A -85,B 0,C 180,E1 -27932.349,E2 -27932.349} C_VEL
LIN {X 0,Y 79.066,Z 193.36,A -85,B 0,C 180,E1 -27936.876,E2 -27936.876} C_VEL
LIN {X 0,Y 82.234,Z 196.266,A -85,B 0,C 180,E1 -27944.241,E2 -27944.241} C_VEL
LIN {X 0,Y 83.993,Z 199.373,A -85,B 0,C 180,E1 -27947.671,E2 -27947.671} C_VEL
LIN {X 0,Y 85.929,Z 201.568,A -85,B 0,C 180,E1 -27950.749,E2 -27950.749} C_VEL
LIN {X 0,Y 89.169,Z 206.439,A -85,B 0,C 180,E1 -27955.273,E2 -27955.273} C_VEL
LIN {X 0,Y 92.011,Z 210.663,A -85,B 0,C 180,E1 -27958.599,E2 -27958.599} C_VEL
LIN {X 0,Y 95.676,Z 216.828,A -85,B 0,C 180,E1 -27962.5,E2 -27962.5} C_VEL
LIN {X 0,Y 100.15,Z 224.884,A -85,B 0,C 180,E1 -27966.582,E2 -27966.582} C_VEL
LIN {X 0,Y 105.79,Z 237.408,A -85,B 0,C 180,E1 -27971.235,E2 -27971.235} C_VEL
LIN {X 0,Y 106.467,Z 239.818,A -85,B 0,C 180,E1 -27971.841,E2 -27971.841} C_VEL
LIN {X 0,Y 102.646,Z 275.109,A -85,B 0,C 180,E1 -27973.933,E2 -27973.933} C_VEL
LIN {X 0,Y 100.263,Z 289.056,A -85,B 0,C 180,E1 -27975.443,E2 -27975.443} C_VEL
LIN {X 0,Y 97.25,Z 301.578,A -85,B 0,C 180,E1 -27977.481,E2 -27977.481} C_VEL
LIN {X 0,Y 93.418,Z 313.702,A -85,B 0,C 180,E1 -27980.257,E2 -27980.257} C_VEL
LIN {X 0,Y 89.03,Z 325.022,A -85,B 0,C 180,E1 -27983.771,E2 -27983.771} C_VEL
LIN {X 0,Y 84.365,Z 335.736,A -85,B 0,C 180,E1 -27988.385,E2 -27988.385} C_VEL
LIN {X 0,Y 80.051,Z 344.917,A -85,B 0,C 180,E1 -27993.778,E2 -27993.778} C_VEL
LIN {X 0,Y 75.914,Z 353.6,A -85,B 0,C 180,E1 -28000.673,E2 -28000.673} C_VEL
LIN {X 0,Y 72.737,Z 360.699,A -85,B 0,C 180,E1 -28008.305,E2 -28008.305} C_VEL
LIN {X 0,Y 70.263,Z 367.322,A -85,B 0,C 180,E1 -28018.032,E2 -28018.032} C_VEL
LIN {X 0,Y 69.396,Z 372.033,A -85,B 0,C 180,E1 -28027.424,E2 -28027.424} C_VEL
LIN {X 0,Y 70.435,Z 376.054,A -85,B 0,C 180,E1 -28038.481,E2 -28038.481} C_VEL
LIN {X 0,Y 73.782,Z 378.535,A -85,B 0,C 180,E1 -28049.02,E2 -28049.02} C_VEL
LIN {X 0,Y 77.235,Z 379.432,A -85,B 0,C 180,E1 -28055.506,E2 -28055.506} C_VEL
LIN {X 0,Y 81.545,Z 379.643,A -85,B 0,C 180,E1 -28061.458,E2 -28061.458} C_VEL
LIN {X 0,Y 86.641,Z 379.249,A -85,B 0,C 180,E1 -28066.767,E2 -28066.767} C_VEL
LIN {X 0,Y 92.397,Z 378.182,A -85,B 0,C 180,E1 -28071.442,E2 -28071.442} C_VEL
LIN {X 0,Y 102.145,Z 375.293,A -85,B 0,C 180,E1 -28077.475,E2 -28077.475} C_VEL
LIN {X 0,Y 112.542,Z 370.894,A -85,B 0,C 180,E1 -28082.29,E2 -28082.29} C_VEL
LIN {X 0,Y 122.235,Z 365.642,A -85,B 0,C 180,E1 -28085.733,E2 -28085.733} C_VEL
LIN {X 0,Y 131.471,Z 359.441,A -85,B 0,C 180,E1 -28088.515,E2 -28088.515} C_VEL
LIN {X 0,Y 141.291,Z 351.386,A -85,B 0,C 180,E1 -28090.925,E2 -28090.925} C_VEL
LIN {X 0,Y 150.465,Z 342.301,A -85,B 0,C 180,E1 -28092.82,E2 -28092.82} C_VEL
LIN {X 0,Y 158.747,Z 332.268,A -85,B 0,C 180,E1 -28094.361,E2 -28094.361} C_VEL
LIN {X 0,Y 166.443,Z 320.758,A -85,B 0,C 180,E1 -28095.641,E2 -28095.641} C_VEL
LIN {X 0,Y 172.748,Z 308.836,A -85,B 0,C 180,E1 -28096.631,E2 -28096.631} C_VEL
LIN {X 0,Y 177.894,Z 296.05,A -85,B 0,C 180,E1 -28097.403,E2 -28097.403} C_VEL
LIN {X 0,Y 178.192,Z 295.183,A -85,B 0,C 180,E1 -28097.544,E2 -28097.544} C_VEL
LIN {X 0,Y 178.123,Z 295.424,A -85,B 0,C 180,E1 -28099.085,E2 -28099.085} C_VEL
LIN {X 0,Y 178.021,Z 295.86,A -85,B 0,C 180,E1 -28099.609,E2 -28099.609} C_VEL
LIN {X 0,Y 177.395,Z 297.733,A -85,B 0,C 180,E1 -28099.93,E2 -28099.93} C_VEL
LIN {X 0,Y 172.528,Z 309.683,A -85,B 0,C 180,E1 -28100.456,E2 -28100.456} C_VEL
LIN {X 0,Y 166.709,Z 320.827,A -85,B 0,C 180,E1 -28101.132,E2 -28101.132} C_VEL
LIN {X 0,Y 159.304,Z 332.176,A -85,B 0,C 180,E1 -28102.107,E2 -28102.107} C_VEL
LIN {X 0,Y 151.154,Z 342.406,A -85,B 0,C 180,E1 -28103.318,E2 -28103.318} C_VEL
LIN {X 0,Y 143.127,Z 350.83,A -85,B 0,C 180,E1 -28104.71,E2 -28104.71} C_VEL
LIN {X 0,Y 133.722,Z 359.147,A -85,B 0,C 180,E1 -28106.684,E2 -28106.684} C_VEL
LIN {X 0,Y 124.5,Z 365.928,A -85,B 0,C 180,E1 -28108.954,E2 -28108.954} C_VEL
LIN {X 0,Y 115.756,Z 371.401,A -85,B 0,C 180,E1 -28111.785,E2 -28111.785} C_VEL
LIN {X 0,Y 107.277,Z 375.809,A -85,B 0,C 180,E1 -28115.021,E2 -28115.021} C_VEL
LIN {X 0,Y 99.34,Z 379.255,A -85,B 0,C 180,E1 -28118.899,E2 -28118.899} C_VEL
LIN {X 0,Y 89.724,Z 382.416,A -85,B 0,C 180,E1 -28125.17,E2 -28125.17} C_VEL
LIN {X 0,Y 81.457,Z 384.128,A -85,B 0,C 180,E1 -28132.843,E2 -28132.843} C_VEL
LIN {X 0,Y 75.077,Z 384.38,A -85,B 0,C 180,E1 -28142.089,E2 -28142.089} C_VEL
LIN {X 0,Y 71.279,Z 383.193,A -85,B 0,C 180,E1 -28152.791,E2 -28152.791} C_VEL
LIN {X 0,Y 70.121,Z 380.551,A -85,B 0,C 180,E1 -28164.244,E2 -28164.244} C_VEL
LIN {X 0,Y 70.289,Z 378.289,A -85,B 0,C 180,E1 -28170.682,E2 -28170.682} C_VEL
LIN {X 0,Y 70.272,Z 374.546,A -85,B 0,C 180,E1 -28178.625,E2 -28178.625} C_VEL
LIN {X 0,Y 71.761,Z 368.248,A -85,B 0,C 180,E1 -28188.556,E2 -28188.556} C_VEL
LIN {X 0,Y 74.547,Z 361.339,A -85,B 0,C 180,E1 -28196.6,E2 -28196.6} C_VEL
LIN {X 0,Y 77.8,Z 354.237,A -85,B 0,C 180,E1 -28202.817,E2 -28202.817} C_VEL
LIN {X 0,Y 81.955,Z 345.669,A -85,B 0,C 180,E1 -28208.438,E2 -28208.438} C_VEL
LIN {X 0,Y 86.827,Z 335.119,A -85,B 0,C 180,E1 -28213.466,E2 -28213.466} C_VEL
LIN {X 0,Y 91.113,Z 324.671,A -85,B 0,C 180,E1 -28217.116,E2 -28217.116} C_VEL
LIN {X 0,Y 95.158,Z 313.244,A -85,B 0,C 180,E1 -28220.015,E2 -28220.015} C_VEL
LIN {X 0,Y 98.826,Z 300.378,A -85,B 0,C 180,E1 -28222.29,E2 -28222.29} C_VEL
LIN {X 0,Y 101.675,Z 286.905,A -85,B 0,C 180,E1 -28223.884,E2 -28223.884} C_VEL
LIN {X 0,Y 103.496,Z 272.448,A -85,B 0,C 180,E1 -28224.931,E2 -28224.931} C_VEL
LIN {X 0,Y 105.884,Z 248.49,A -85,B 0,C 180,E1 -28226.369,E2 -28226.369} C_VEL
LIN {X 0,Y 105.675,Z 244.886,A -85,B 0,C 180,E1 -28226.864,E2 -28226.864} C_VEL
LIN {X 0,Y 102.442,Z 233.41,A -85,B 0,C 180,E1 -28229.887,E2 -28229.887} C_VEL
LIN {X 0,Y 99.054,Z 223.641,A -85,B 0,C 180,E1 -28233.142,E2 -28233.142} C_VEL
LIN {X 0,Y 94.416,Z 214.868,A -85,B 0,C 180,E1 -28237.603,E2 -28237.603} C_VEL
LIN {X 0,Y 89.962,Z 207.476,A -85,B 0,C 180,E1 -28242.67,E2 -28242.67} C_VEL
LIN {X 0,Y 88.219,Z 204.793,A -85,B 0,C 180,E1 -28244.881,E2 -28244.881} C_VEL
LIN {X 0,Y 85.647,Z 200.834,A -85,B 0,C 180,E1 -28248.618,E2 -28248.618} C_VEL
LIN {X 0,Y 82.898,Z 196.855,A -85,B 0,C 180,E1 -28253.456,E2 -28253.456} C_VEL
LIN {X 0,Y 82.25,Z 195.718,A -85,B 0,C 180,E1 -28254.788,E2 -28254.788} C_VEL
LIN {X 0,Y 80.504,Z 194.146,A -85,B 0,C 180,E1 -28258.423,E2 -28258.423} C_VEL
LIN {X 0,Y 79.412,Z 193.515,A -85,B 0,C 180,E1 -28261.066,E2 -28261.066} C_VEL
LIN {X 0,Y 77.955,Z 194.298,A -85,B 0,C 180,E1 -28264.736,E2 -28264.736} C_VEL
LIN {X 0,Y 75.895,Z 196.736,A -85,B 0,C 180,E1 -28271.493,E2 -28271.493} C_VEL
LIN {X 0,Y 75.562,Z 196.909,A -85,B 0,C 180,E1 -28273.545,E2 -28273.545} C_VEL
LIN {X 0,Y 75.858,Z 197.184,A -85,B 0,C 180,E1 -28287.593,E2 -28287.593} C_VEL
LIN {X 0,Y 76.63,Z 197.676,A -85,B 0,C 180,E1 -28291.437,E2 -28291.437} C_VEL
LIN {X 0,Y 77.888,Z 200.588,A -85,B 0,C 180,E1 -28296.71,E2 -28296.71} C_VEL
LIN {X 0,Y 80.285,Z 203.001,A -85,B 0,C 180,E1 -28302.742,E2 -28302.742} C_VEL
LIN {X 0,Y 82.348,Z 206.306,A -85,B 0,C 180,E1 -28306.944,E2 -28306.944} C_VEL
LIN {X 0,Y 83.62,Z 207.978,A -85,B 0,C 180,E1 -28309.145,E2 -28309.145} C_VEL
LIN {X 0,Y 86.73,Z 212.911,A -85,B 0,C 180,E1 -28313.919,E2 -28313.919} C_VEL
LIN {X 0,Y 90.107,Z 218.272,A -85,B 0,C 180,E1 -28318.149,E2 -28318.149} C_VEL
LIN {X 0,Y 95.782,Z 228.885,A -85,B 0,C 180,E1 -28324.247,E2 -28324.247} C_VEL
LIN {X 0,Y 101.123,Z 241.197,A -85,B 0,C 180,E1 -28329.131,E2 -28329.131} C_VEL
LIN {X 0,Y 97.439,Z 274.794,A -85,B 0,C 180,E1 -28331.178,E2 -28331.178} C_VEL
LIN {X 0,Y 95.017,Z 288.387,A -85,B 0,C 180,E1 -28332.618,E2 -28332.618} C_VEL
LIN {X 0,Y 91.799,Z 301.406,A -85,B 0,C 180,E1 -28334.744,E2 -28334.744} C_VEL
LIN {X 0,Y 87.707,Z 313.695,A -85,B 0,C 180,E1 -28337.585,E2 -28337.585} C_VEL
LIN {X 0,Y 82.786,Z 325.727,A -85,B 0,C 180,E1 -28341.459,E2 -28341.459} C_VEL
LIN {X 0,Y 78.25,Z 335.51,A -85,B 0,C 180,E1 -28345.856,E2 -28345.856} C_VEL
LIN {X 0,Y 73.761,Z 344.499,A -85,B 0,C 180,E1 -28351.368,E2 -28351.368} C_VEL
LIN {X 0,Y 69.243,Z 353.329,A -85,B 0,C 180,E1 -28358.797,E2 -28358.797} C_VEL
LIN {X 0,Y 65.977,Z 360.097,A -85,B 0,C 180,E1 -28366.538,E2 -28366.538} C_VEL
LIN {X 0,Y 63.395,Z 366.475,A -85,B 0,C 180,E1 -28376.328,E2 -28376.328} C_VEL
LIN {X 0,Y 62.299,Z 371.894,A -85,B 0,C 180,E1 -28387.851,E2 -28387.851} C_VEL
LIN {X 0,Y 63.682,Z 376.198,A -85,B 0,C 180,E1 -28400.588,E2 -28400.588} C_VEL
LIN {X 0,Y 66.026,Z 378.067,A -85,B 0,C 180,E1 -28408.387,E2 -28408.387} C_VEL
LIN {X 0,Y 69.865,Z 379.418,A -85,B 0,C 180,E1 -28416.277,E2 -28416.277} C_VEL
LIN {X 0,Y 75.1,Z 380.02,A -85,B 0,C 180,E1 -28423.698,E2 -28423.698} C_VEL
LIN {X 0,Y 81.427,Z 379.739,A -85,B 0,C 180,E1 -28430.063,E2 -28430.063} C_VEL
LIN {X 0,Y 91.475,Z 377.943,A -85,B 0,C 180,E1 -28437.231,E2 -28437.231} C_VEL
LIN {X 0,Y 101.619,Z 374.874,A -85,B 0,C 180,E1 -28442.427,E2 -28442.427} C_VEL
LIN {X 0,Y 109.458,Z 371.686,A -85,B 0,C 180,E1 -28445.585,E2 -28445.585} C_VEL
LIN {X 0,Y 121.061,Z 365.692,A -85,B 0,C 180,E1 -28449.269,E2 -28449.269} C_VEL
LIN {X 0,Y 130.828,Z 359.296,A -85,B 0,C 180,E1 -28451.828,E2 -28451.828} C_VEL
LIN {X 0,Y 140.753,Z 351.385,A -85,B 0,C 180,E1 -28453.933,E2 -28453.933} C_VEL
LIN {X 0,Y 149.544,Z 342.895,A -85,B 0,C 180,E1 -28455.538,E2 -28455.538} C_VEL
LIN {X 0,Y 157.931,Z 333.038,A -85,B 0,C 180,E1 -28456.905,E2 -28456.905} C_VEL
LIN {X 0,Y 165.431,Z 322.171,A -85,B 0,C 180,E1 -28458.018,E2 -28458.018} C_VEL
LIN {X 0,Y 166.858,Z 319.861,A -85,B 0,C 180,E1 -28458.226,E2 -28458.226} C_VEL
LIN {X 0,Y 166.232,Z 320.952,A -85,B 0,C 180,E1 -28458.676,E2 -28458.676} C_VEL
LIN {X 0,Y 158.494,Z 332.514,A -85,B 0,C 180,E1 -28459.558,E2 -28459.558} C_VEL
LIN {X 0,Y 150.191,Z 342.639,A -85,B 0,C 180,E1 -28460.625,E2 -28460.625} C_VEL
LIN {X 0,Y 140.351,Z 352.411,A -85,B 0,C 180,E1 -28462.119,E2 -28462.119} C_VEL
LIN {X 0,Y 130.724,Z 360.326,A -85,B 0,C 180,E1 -28463.937,E2 -28463.937} C_VEL
LIN {X 0,Y 121.252,Z 366.814,A -85,B 0,C 180,E1 -28466.046,E2 -28466.046} C_VEL
LIN {X 0,Y 112.203,Z 372.049,A -85,B 0,C 180,E1 -28468.724,E2 -28468.724} C_VEL
LIN {X 0,Y 103.372,Z 376.235,A -85,B 0,C 180,E1 -28471.801,E2 -28471.801} C_VEL
LIN {X 0,Y 95.04,Z 379.453,A -85,B 0,C 180,E1 -28475.564,E2 -28475.564} C_VEL
LIN {X 0,Y 84.83,Z 382.409,A -85,B 0,C 180,E1 -28481.782,E2 -28481.782} C_VEL
LIN {X 0,Y 75.902,Z 383.887,A -85,B 0,C 180,E1 -28489.594,E2 -28489.594} C_VEL
LIN {X 0,Y 68.867,Z 383.919,A -85,B 0,C 180,E1 -28499.315,E2 -28499.315} C_VEL
LIN {X 0,Y 64.529,Z 382.568,A -85,B 0,C 180,E1 -28510.925,E2 -28510.925} C_VEL
LIN {X 0,Y 63.459,Z 381.331,A -85,B 0,C 180,E1 -28517.199,E2 -28517.199} C_VEL
LIN {X 0,Y 63.276,Z 378.124,A -85,B 0,C 180,E1 -28528.566,E2 -28528.566} C_VEL
LIN {X 0,Y 63.122,Z 374.93,A -85,B 0,C 180,E1 -28536.389,E2 -28536.389} C_VEL
LIN {X 0,Y 64.338,Z 368.901,A -85,B 0,C 180,E1 -28547.478,E2 -28547.478} C_VEL
LIN {X 0,Y 67.05,Z 362.24,A -85,B 0,C 180,E1 -28556.45,E2 -28556.45} C_VEL
LIN {X 0,Y 71.113,Z 353.916,A -85,B 0,C 180,E1 -28564.626,E2 -28564.626} C_VEL
LIN {X 0,Y 75.54,Z 345.374,A -85,B 0,C 180,E1 -28570.632,E2 -28570.632} C_VEL
LIN {X 0,Y 80.588,Z 335.078,A -85,B 0,C 180,E1 -28575.826,E2 -28575.826} C_VEL
LIN {X 0,Y 85.234,Z 324.413,A -85,B 0,C 180,E1 -28579.7,E2 -28579.7} C_VEL
LIN {X 0,Y 89.5,Z 313.019,A -85,B 0,C 180,E1 -28582.657,E2 -28582.657} C_VEL
LIN {X 0,Y 93.333,Z 300.172,A -85,B 0,C 180,E1 -28584.97,E2 -28584.97} C_VEL
LIN {X 0,Y 96.239,Z 287.094,A -85,B 0,C 180,E1 -28586.549,E2 -28586.549} C_VEL
LIN {X 0,Y 98.086,Z 273.737,A -85,B 0,C 180,E1 -28587.54,E2 -28587.54} C_VEL
LIN {X 0,Y 100.654,Z 248.648,A -85,B 0,C 180,E1 -28589.095,E2 -28589.095} C_VEL
LIN {X 0,Y 100.214,Z 245.771,A -85,B 0,C 180,E1 -28589.692,E2 -28589.692} C_VEL
LIN {X 0,Y 97.087,Z 234.539,A -85,B 0,C 180,E1 -28593.003,E2 -28593.003} C_VEL
LIN {X 0,Y 94.719,Z 227.641,A -85,B 0,C 180,E1 -28595.547,E2 -28595.547} C_VEL
LIN {X 0,Y 90.473,Z 219.253,A -85,B 0,C 180,E1 -28600.227,E2 -28600.227} C_VEL
LIN {X 0,Y 86.496,Z 212.296,A -85,B 0,C 180,E1 -28605.326,E2 -28605.326} C_VEL
LIN {X 0,Y 82.529,Z 205.964,A -85,B 0,C 180,E1 -28611.726,E2 -28611.726} C_VEL
LIN {X 0,Y 80.199,Z 202.203,A -85,B 0,C 180,E1 -28616.543,E2 -28616.543} C_VEL
LIN {X 0,Y 78.197,Z 199.676,A -85,B 0,C 180,E1 -28621.687,E2 -28621.687} C_VEL
LIN {X 0,Y 77.33,Z 197.384,A -85,B 0,C 180,E1 -28625.212,E2 -28625.212} C_VEL
LIN {X 0,Y 75.562,Z 196.909,A -85,B 0,C 180,E1 -28633.545,E2 -28633.545} C_VEL
LIN {X 0,Y 75.142,Z 197.583,A -85,B 0,C 180,E1 -28637.993,E2 -28637.993} C_VEL
LIN {X 0,Y 74.945,Z 199.463,A -85,B 0,C 180,E1 -28642.307,E2 -28642.307} C_VEL
LIN {X 0,Y 75.916,Z 206.332,A -85,B 0,C 180,E1 -28653.446,E2 -28653.446} C_VEL
LIN {X 0,Y 76.642,Z 207.642,A -85,B 0,C 180,E1 -28656.28,E2 -28656.28} C_VEL
LIN {X 0,Y 78.368,Z 209.545,A -85,B 0,C 180,E1 -28661.056,E2 -28661.056} C_VEL
LIN {X 0,Y 80.701,Z 213.228,A -85,B 0,C 180,E1 -28666.187,E2 -28666.187} C_VEL
LIN {X 0,Y 83.659,Z 218.208,A -85,B 0,C 180,E1 -28671.426,E2 -28671.426} C_VEL
LIN {X 0,Y 86.78,Z 223.499,A -85,B 0,C 180,E1 -28675.906,E2 -28675.906} C_VEL
LIN {X 0,Y 91.867,Z 233.56,A -85,B 0,C 180,E1 -28682.017,E2 -28682.017} C_VEL
LIN {X 0,Y 96.005,Z 243.665,A -85,B 0,C 180,E1 -28686.366,E2 -28686.366} C_VEL
LIN {X 0,Y 92.141,Z 275.844,A -85,B 0,C 180,E1 -28688.275,E2 -28688.275} C_VEL
LIN {X 0,Y 89.429,Z 290.246,A -85,B 0,C 180,E1 -28689.898,E2 -28689.898} C_VEL
LIN {X 0,Y 85.834,Z 303.265,A -85,B 0,C 180,E1 -28692.122,E2 -28692.122} C_VEL
LIN {X 0,Y 81.529,Z 315.205,A -85,B 0,C 180,E1 -28695.016,E2 -28695.016} C_VEL
LIN {X 0,Y 76.57,Z 326.623,A -85,B 0,C 180,E1 -28698.902,E2 -28698.902} C_VEL
LIN {X 0,Y 71.064,Z 337.655,A -85,B 0,C 180,E1 -28704.328,E2 -28704.328} C_VEL
LIN {X 0,Y 65.531,Z 347.859,A -85,B 0,C 180,E1 -28711.54,E2 -28711.54} C_VEL
LIN {X 0,Y 61.008,Z 356.1,A -85,B 0,C 180,E1 -28719.954,E2 -28719.954} C_VEL
LIN {X 0,Y 57.95,Z 362.376,A -85,B 0,C 180,E1 -28728.741,E2 -28728.741} C_VEL
LIN {X 0,Y 55.653,Z 368.468,A -85,B 0,C 180,E1 -28740.345,E2 -28740.345} C_VEL
LIN {X 0,Y 55.52,Z 373.73,A -85,B 0,C 180,E1 -28754.257,E2 -28754.257} C_VEL
LIN {X 0,Y 58.28,Z 377.359,A -85,B 0,C 180,E1 -28767.587,E2 -28767.587} C_VEL
LIN {X 0,Y 61.686,Z 379.016,A -85,B 0,C 180,E1 -28775.715,E2 -28775.715} C_VEL
LIN {X 0,Y 66.154,Z 380.006,A -85,B 0,C 180,E1 -28782.977,E2 -28782.977} C_VEL
LIN {X 0,Y 71.53,Z 380.375,A -85,B 0,C 180,E1 -28789.292,E2 -28789.292} C_VEL
LIN {X 0,Y 77.886,Z 380.096,A -85,B 0,C 180,E1 -28794.826,E2 -28794.826} C_VEL
LIN {X 0,Y 85.693,Z 378.949,A -85,B 0,C 180,E1 -28800.003,E2 -28800.003} C_VEL
LIN {X 0,Y 94.184,Z 376.908,A -85,B 0,C 180,E1 -28804.282,E2 -28804.282} C_VEL
LIN {X 0,Y 103.092,Z 373.936,A -85,B 0,C 180,E1 -28807.839,E2 -28807.839} C_VEL
LIN {X 0,Y 114.716,Z 368.834,A -85,B 0,C 180,E1 -28811.4,E2 -28811.4} C_VEL
LIN {X 0,Y 124.918,Z 363.059,A -85,B 0,C 180,E1 -28813.944,E2 -28813.944} C_VEL
LIN {X 0,Y 135.306,Z 355.757,A -85,B 0,C 180,E1 -28816.032,E2 -28816.032} C_VEL
LIN {X 0,Y 145.086,Z 347.341,A -85,B 0,C 180,E1 -28817.665,E2 -28817.665} C_VEL
LIN {X 0,Y 146.417,Z 346.066,A -85,B 0,C 180,E1 -28817.879,E2 -28817.879} C_VEL
LIN {X 0,Y 144.524,Z 347.943,A -85,B 0,C 180,E1 -28818.507,E2 -28818.507} C_VEL
LIN {X 0,Y 134.586,Z 356.644,A -85,B 0,C 180,E1 -28819.951,E2 -28819.951} C_VEL
LIN {X 0,Y 124.789,Z 363.734,A -85,B 0,C 180,E1 -28821.674,E2 -28821.674} C_VEL
LIN {X 0,Y 115.219,Z 369.479,A -85,B 0,C 180,E1 -28823.796,E2 -28823.796} C_VEL
LIN {X 0,Y 105.908,Z 374.092,A -85,B 0,C 180,E1 -28826.376,E2 -28826.376} C_VEL
LIN {X 0,Y 96.861,Z 377.74,A -85,B 0,C 180,E1 -28829.456,E2 -28829.456} C_VEL
LIN {X 0,Y 85.561,Z 381.215,A -85,B 0,C 180,E1 -28834.77,E2 -28834.77} C_VEL
LIN {X 0,Y 75.282,Z 383.159,A -85,B 0,C 180,E1 -28841.677,E2 -28841.677} C_VEL
LIN {X 0,Y 66.494,Z 383.706,A -85,B 0,C 180,E1 -28850.638,E2 -28850.638} C_VEL
LIN {X 0,Y 62.851,Z 383.455,A -85,B 0,C 180,E1 -28856.002,E2 -28856.002} C_VEL
LIN {X 0,Y 57.871,Z 381.865,A -85,B 0,C 180,E1 -28868.629,E2 -28868.629} C_VEL
LIN {X 0,Y 56.115,Z 378.795,A -85,B 0,C 180,E1 -28882.801,E2 -28882.801} C_VEL
LIN {X 0,Y 56.228,Z 376.619,A -85,B 0,C 180,E1 -28889.996,E2 -28889.996} C_VEL
LIN {X 0,Y 56.282,Z 372.19,A -85,B 0,C 180,E1 -28900.791,E2 -28900.791} C_VEL
LIN {X 0,Y 57.983,Z 366.476,A -85,B 0,C 180,E1 -28911.319,E2 -28911.319} C_VEL
LIN {X 0,Y 61.452,Z 359.273,A -85,B 0,C 180,E1 -28920.969,E2 -28920.969} C_VEL
LIN {X 0,Y 66.274,Z 350.255,A -85,B 0,C 180,E1 -28929.509,E2 -28929.509} C_VEL
LIN {X 0,Y 71.169,Z 341.405,A -85,B 0,C 180,E1 -28935.337,E2 -28935.337} C_VEL
LIN {X 0,Y 76.469,Z 330.882,A -85,B 0,C 180,E1 -28940.218,E2 -28940.218} C_VEL
LIN {X 0,Y 81.463,Z 319.409,A -85,B 0,C 180,E1 -28943.974,E2 -28943.974} C_VEL
LIN {X 0,Y 85.726,Z 307.729,A -85,B 0,C 180,E1 -28946.631,E2 -28946.631} C_VEL
LIN {X 0,Y 89.274,Z 295.079,A -85,B 0,C 180,E1 -28948.608,E2 -28948.608} C_VEL
LIN {X 0,Y 92.052,Z 281.38,A -85,B 0,C 180,E1 -28949.966,E2 -28949.966} C_VEL
LIN {X 0,Y 95.611,Z 249.546,A -85,B 0,C 180,E1 -28951.998,E2 -28951.998} C_VEL
LIN {X 0,Y 92.873,Z 238.848,A -85,B 0,C 180,E1 -28955.313,E2 -28955.313} C_VEL
LIN {X 0,Y 90.716,Z 232.006,A -85,B 0,C 180,E1 -28957.998,E2 -28957.998} C_VEL
LIN {X 0,Y 86.975,Z 224.116,A -85,B 0,C 180,E1 -28962.678,E2 -28962.678} C_VEL
LIN {X 0,Y 83.146,Z 217.001,A -85,B 0,C 180,E1 -28968.332,E2 -28968.332} C_VEL
LIN {X 0,Y 80.25,Z 212.129,A -85,B 0,C 180,E1 -28973.712,E2 -28973.712} C_VEL
LIN {X 0,Y 78.23,Z 208.661,A -85,B 0,C 180,E1 -28978.388,E2 -28978.388} C_VEL
LIN {X 0,Y 76.405,Z 205.762,A -85,B 0,C 180,E1 -28984.071,E2 -28984.071} C_VEL
LIN {X 0,Y 75.984,Z 204.348,A -85,B 0,C 180,E1 -28986.202,E2 -28986.202} C_VEL
LIN {X 0,Y 74.186,Z 203.906,A -85,B 0,C 180,E1 -28998.684,E2 -28998.684} C_VEL
LIN {X 0,Y 75.127,Z 204.377,A -85,B 0,C 180,E1 -29009.411,E2 -29009.411} C_VEL
LIN {X 0,Y 76.642,Z 207.642,A -85,B 0,C 180,E1 -29016.28,E2 -29016.28} C_VEL
LIN {X 0,Y 77.44,Z 209.152,A -85,B 0,C 180,E1 -29018.899,E2 -29018.899} C_VEL
LIN {X 0,Y 78.529,Z 212.635,A -85,B 0,C 180,E1 -29022.323,E2 -29022.323} C_VEL
LIN {X 0,Y 82.031,Z 225.828,A -85,B 0,C 180,E1 -29030.994,E2 -29030.994} C_VEL
LIN {X 0,Y 83.31,Z 228.263,A -85,B 0,C 180,E1 -29033.071,E2 -29033.071} C_VEL
LIN {X 0,Y 87.354,Z 236.701,A -85,B 0,C 180,E1 -29038.709,E2 -29038.709} C_VEL
LIN {X 0,Y 90.079,Z 243.468,A -85,B 0,C 180,E1 -29042.091,E2 -29042.091} C_VEL
LIN {X 0,Y 90.959,Z 245.758,A -85,B 0,C 180,E1 -29043.119,E2 -29043.119} C_VEL
LIN {X 0,Y 87.836,Z 272.612,A -85,B 0,C 180,E1 -29044.777,E2 -29044.777} C_VEL
LIN {X 0,Y 85.412,Z 286.128,A -85,B 0,C 180,E1 -29045.993,E2 -29045.993} C_VEL
LIN {X 0,Y 82.163,Z 298.684,A -85,B 0,C 180,E1 -29047.87,E2 -29047.87} C_VEL
LIN {X 0,Y 78.216,Z 310.245,A -85,B 0,C 180,E1 -29050.312,E2 -29050.312} C_VEL
LIN {X 0,Y 73.208,Z 321.936,A -85,B 0,C 180,E1 -29053.729,E2 -29053.729} C_VEL
LIN {X 0,Y 68.056,Z 332.24,A -85,B 0,C 180,E1 -29058.084,E2 -29058.084} C_VEL
LIN {X 0,Y 62.251,Z 342.518,A -85,B 0,C 180,E1 -29064.335,E2 -29064.335} C_VEL
LIN {X 0,Y 57.305,Z 350.9,A -85,B 0,C 180,E1 -29071.713,E2 -29071.713} C_VEL
LIN {X 0,Y 52.771,Z 358.721,A -85,B 0,C 180,E1 -29081.528,E2 -29081.528} C_VEL
LIN {X 0,Y 49.621,Z 365.102,A -85,B 0,C 180,E1 -29092.926,E2 -29092.926} C_VEL
LIN {X 0,Y 48.175,Z 370.33,A -85,B 0,C 180,E1 -29105.706,E2 -29105.706} C_VEL
LIN {X 0,Y 49.348,Z 375.094,A -85,B 0,C 180,E1 -29121.288,E2 -29121.288} C_VEL
LIN {X 0,Y 53.9,Z 378.455,A -85,B 0,C 180,E1 -29135.896,E2 -29135.896} C_VEL
LIN {X 0,Y 60.243,Z 380.153,A -85,B 0,C 180,E1 -29146.511,E2 -29146.511} C_VEL
LIN {X 0,Y 67.094,Z 380.743,A -85,B 0,C 180,E1 -29153.991,E2 -29153.991} C_VEL
LIN {X 0,Y 77.34,Z 380.193,A -85,B 0,C 180,E1 -29161.54,E2 -29161.54} C_VEL
LIN {X 0,Y 84.73,Z 379.069,A -85,B 0,C 180,E1 -29165.501,E2 -29165.501} C_VEL
LIN {X 0,Y 96.407,Z 376.114,A -85,B 0,C 180,E1 -29170.204,E2 -29170.204} C_VEL
LIN {X 0,Y 108.559,Z 371.64,A -85,B 0,C 180,E1 -29173.804,E2 -29173.804} C_VEL
LIN {X 0,Y 119.235,Z 366.426,A -85,B 0,C 180,E1 -29176.281,E2 -29176.281} C_VEL
LIN {X 0,Y 125.269,Z 362.867,A -85,B 0,C 180,E1 -29177.486,E2 -29177.486} C_VEL
LIN {X 0,Y 125.694,Z 362.64,A -85,B 0,C 180,E1 -29178.091,E2 -29178.091} C_VEL
LIN {X 0,Y 115.77,Z 368.549,A -85,B 0,C 180,E1 -29179.782,E2 -29179.782} C_VEL
LIN {X 0,Y 106.147,Z 373.27,A -85,B 0,C 180,E1 -29182.031,E2 -29182.031} C_VEL
LIN {X 0,Y 96.665,Z 377.007,A -85,B 0,C 180,E1 -29184.653,E2 -29184.653} C_VEL
LIN {X 0,Y 87.541,Z 379.83,A -85,B 0,C 180,E1 -29187.974,E2 -29187.974} C_VEL
LIN {X 0,Y 76.096,Z 382.282,A -85,B 0,C 180,E1 -29193.771,E2 -29193.771} C_VEL
LIN {X 0,Y 65.715,Z 383.327,A -85,B 0,C 180,E1 -29201.523,E2 -29201.523} C_VEL
LIN {X 0,Y 57.094,Z 382.926,A -85,B 0,C 180,E1 -29212.009,E2 -29212.009} C_VEL
LIN {X 0,Y 51.335,Z 381.126,A -85,B 0,C 180,E1 -29225.746,E2 -29225.746} C_VEL
LIN {X 0,Y 49.138,Z 377.865,A -85,B 0,C 180,E1 -29241.772,E2 -29241.772} C_VEL
LIN {X 0,Y 49.16,Z 375.542,A -85,B 0,C 180,E1 -29249.995,E2 -29249.995} C_VEL
LIN {X 0,Y 49.334,Z 370.912,A -85,B 0,C 180,E1 -29262.334,E2 -29262.334} C_VEL
LIN {X 0,Y 51.426,Z 364.966,A -85,B 0,C 180,E1 -29274.199,E2 -29274.199} C_VEL
LIN {X 0,Y 55.485,Z 357.516,A -85,B 0,C 180,E1 -29284.744,E2 -29284.744} C_VEL
LIN {X 0,Y 59.933,Z 349.842,A -85,B 0,C 180,E1 -29292.392,E2 -29292.392} C_VEL
LIN {X 0,Y 65.425,Z 340.587,A -85,B 0,C 180,E1 -29298.753,E2 -29298.753} C_VEL
LIN {X 0,Y 71.406,Z 329.256,A -85,B 0,C 180,E1 -29304.042,E2 -29304.042} C_VEL
LIN {X 0,Y 76.838,Z 317.334,A -85,B 0,C 180,E1 -29307.779,E2 -29307.779} C_VEL
LIN {X 0,Y 81.339,Z 305.017,A -85,B 0,C 180,E1 -29310.388,E2 -29310.388} C_VEL
LIN {X 0,Y 85.071,Z 291.568,A -85,B 0,C 180,E1 -29312.309,E2 -29312.309} C_VEL
LIN {X 0,Y 87.431,Z 278.945,A -85,B 0,C 180,E1 -29313.43,E2 -29313.43} C_VEL
LIN {X 0,Y 90.708,Z 251.246,A -85,B 0,C 180,E1 -29315.124,E2 -29315.124} C_VEL
LIN {X 0,Y 88.229,Z 240.998,A -85,B 0,C 180,E1 -29318.686,E2 -29318.686} C_VEL
LIN {X 0,Y 86.893,Z 236.367,A -85,B 0,C 180,E1 -29320.661,E2 -29320.661} C_VEL
LIN {X 0,Y 83.408,Z 228.609,A -85,B 0,C 180,E1 -29325.613,E2 -29325.613} C_VEL
LIN {X 0,Y 80.596,Z 222.942,A -85,B 0,C 180,E1 -29330.453,E2 -29330.453} C_VEL
LIN {X 0,Y 77.866,Z 217.977,A -85,B 0,C 180,E1 -29336.192,E2 -29336.192} C_VEL
LIN {X 0,Y 76.472,Z 215.209,A -85,B 0,C 180,E1 -29339.997,E2 -29339.997} C_VEL
LIN {X 0,Y 74.809,Z 212.095,A -85,B 0,C 180,E1 -29346.185,E2 -29346.185} C_VEL
LIN {X 0,Y 74.529,Z 211.267,A -85,B 0,C 180,E1 -29347.65,E2 -29347.65} C_VEL
LIN {X 0,Y 73.204,Z 210.85,A -85,B 0,C 180,E1 -29356.736,E2 -29356.736} C_VEL
LIN {X 0,Y 73.931,Z 211.429,A -85,B 0,C 180,E1 -29368.763,E2 -29368.763} C_VEL
LIN {X 0,Y 75.44,Z 214.746,A -85,B 0,C 180,E1 -29375.972,E2 -29375.972} C_VEL
LIN {X 0,Y 76.603,Z 216.239,A -85,B 0,C 180,E1 -29379.529,E2 -29379.529} C_VEL
LIN {X 0,Y 79.123,Z 220.594,A -85,B 0,C 180,E1 -29385.603,E2 -29385.603} C_VEL
LIN {X 0,Y 82.452,Z 226.505,A -85,B 0,C 180,E1 -29391.678,E2 -29391.678} C_VEL
LIN {X 0,Y 83.31,Z 228.263,A -85,B 0,C 180,E1 -29393.071,E2 -29393.071} C_VEL
LIN {X 0,Y 84.217,Z 230.52,A -85,B 0,C 180,E1 -29394.53,E2 -29394.53} C_VEL
LIN {X 0,Y 84.772,Z 234.67,A -85,B 0,C 180,E1 -29395.889,E2 -29395.889} C_VEL
LIN {X 0,Y 85.16,Z 243.85,A -85,B 0,C 180,E1 -29397.901,E2 -29397.901} C_VEL
LIN {X 0,Y 85.981,Z 247.328,A -85,B 0,C 180,E1 -29399.243,E2 -29399.243} C_VEL
LIN {X 0,Y 86.324,Z 248.284,A -85,B 0,C 180,E1 -29399.704,E2 -29399.704} C_VEL
LIN {X 0,Y 82.704,Z 276.2,A -85,B 0,C 180,E1 -29401.318,E2 -29401.318} C_VEL
LIN {X 0,Y 79.771,Z 290.309,A -85,B 0,C 180,E1 -29402.832,E2 -29402.832} C_VEL
LIN {X 0,Y 76.121,Z 302.546,A -85,B 0,C 180,E1 -29404.802,E2 -29404.802} C_VEL
LIN {X 0,Y 71.395,Z 314.544,A -85,B 0,C 180,E1 -29407.58,E2 -29407.58} C_VEL
LIN {X 0,Y 65.918,Z 325.87,A -85,B 0,C 180,E1 -29411.35,E2 -29411.35} C_VEL
LIN {X 0,Y 60.098,Z 336.311,A -85,B 0,C 180,E1 -29416.478,E2 -29416.478} C_VEL
LIN {X 0,Y 54.747,Z 344.917,A -85,B 0,C 180,E1 -29422.629,E2 -29422.629} C_VEL
LIN {X 0,Y 49.21,Z 353.427,A -85,B 0,C 180,E1 -29431.569,E2 -29431.569} C_VEL
LIN {X 0,Y 44.912,Z 360.399,A -85,B 0,C 180,E1 -29442.326,E2 -29442.326} C_VEL
LIN {X 0,Y 41.679,Z 367.213,A -85,B 0,C 180,E1 -29457.633,E2 -29457.633} C_VEL
LIN {X 0,Y 41.191,Z 372.117,A -85,B 0,C 180,E1 -29473.046,E2 -29473.046} C_VEL
LIN {X 0,Y 44.544,Z 376.688,A -85,B 0,C 180,E1 -29491.755,E2 -29491.755} C_VEL
LIN {X 0,Y 50.819,Z 379.412,A -85,B 0,C 180,E1 -29505.5,E2 -29505.5} C_VEL
LIN {X 0,Y 56.627,Z 380.552,A -85,B 0,C 180,E1 -29513.192,E2 -29513.192} C_VEL
LIN {X 0,Y 64.022,Z 381.107,A -85,B 0,C 180,E1 -29520.003,E2 -29520.003} C_VEL
LIN {X 0,Y 72.584,Z 380.826,A -85,B 0,C 180,E1 -29525.56,E2 -29525.56} C_VEL
LIN {X 0,Y 81.653,Z 379.686,A -85,B 0,C 180,E1 -29529.915,E2 -29529.915} C_VEL
LIN {X 0,Y 94.286,Z 376.834,A -85,B 0,C 180,E1 -29534.291,E2 -29534.291} C_VEL
LIN {X 0,Y 106.484,Z 372.633,A -85,B 0,C 180,E1 -29537.384,E2 -29537.384} C_VEL
LIN {X 0,Y 104.707,Z 373.434,A -85,B 0,C 180,E1 -29538.197,E2 -29538.197} C_VEL
LIN {X 0,Y 93.937,Z 377.372,A -85,B 0,C 180,E1 -29540.732,E2 -29540.732} C_VEL
LIN {X 0,Y 84.449,Z 379.977,A -85,B 0,C 180,E1 -29543.724,E2 -29543.724} C_VEL
LIN {X 0,Y 72.383,Z 382.201,A -85,B 0,C 180,E1 -29549.083,E2 -29549.083} C_VEL
LIN {X 0,Y 61.233,Z 382.971,A -85,B 0,C 180,E1 -29556.535,E2 -29556.535} C_VEL
LIN {X 0,Y 51.679,Z 382.355,A -85,B 0,C 180,E1 -29567.153,E2 -29567.153} C_VEL
LIN {X 0,Y 44.972,Z 380.38,A -85,B 0,C 180,E1 -29582.036,E2 -29582.036} C_VEL
LIN {X 0,Y 43.044,Z 378.818,A -85,B 0,C 180,E1 -29590.935,E2 -29590.935} C_VEL
LIN {X 0,Y 42.117,Z 375.727,A -85,B 0,C 180,E1 -29605.208,E2 -29605.208} C_VEL
LIN {X 0,Y 42.102,Z 374.41,A -85,B 0,C 180,E1 -29609.994,E2 -29609.994} C_VEL
LIN {X 0,Y 42.445,Z 369.56,A -85,B 0,C 180,E1 -29624.375,E2 -29624.375} C_VEL
LIN {X 0,Y 45.04,Z 363.37,A -85,B 0,C 180,E1 -29637.906,E2 -29637.906} C_VEL
LIN {X 0,Y 49.819,Z 355.618,A -85,B 0,C 180,E1 -29649.401,E2 -29649.401} C_VEL
LIN {X 0,Y 54.92,Z 347.63,A -85,B 0,C 180,E1 -29657.37,E2 -29657.37} C_VEL
LIN {X 0,Y 60.962,Z 337.94,A -85,B 0,C 180,E1 -29663.796,E2 -29663.796} C_VEL
LIN {X 0,Y 66.252,Z 328.49,A -85,B 0,C 180,E1 -29668.058,E2 -29668.058} C_VEL
LIN {X 0,Y 71.864,Z 316.803,A -85,B 0,C 180,E1 -29671.655,E2 -29671.655} C_VEL
LIN {X 0,Y 76.599,Z 304.476,A -85,B 0,C 180,E1 -29674.191,E2 -29674.191} C_VEL
LIN {X 0,Y 80.326,Z 291.657,A -85,B 0,C 180,E1 -29675.969,E2 -29675.969} C_VEL
LIN {X 0,Y 83,Z 277.975,A -85,B 0,C 180,E1 -29677.118,E2 -29677.118} C_VEL
LIN {X 0,Y 86.053,Z 252.794,A -85,B 0,C 180,E1 -29678.669,E2 -29678.669} C_VEL
LIN {X 0,Y 83.597,Z 241.858,A -85,B 0,C 180,E1 -29682.88,E2 -29682.88} C_VEL
LIN {X 0,Y 80.739,Z 234.671,A -85,B 0,C 180,E1 -29687.583,E2 -29687.583} C_VEL
LIN {X 0,Y 78.091,Z 228.77,A -85,B 0,C 180,E1 -29692.819,E2 -29692.819} C_VEL
LIN {X 0,Y 75.638,Z 223.787,A -85,B 0,C 180,E1 -29698.834,E2 -29698.834} C_VEL
LIN {X 0,Y 74.609,Z 221.56,A -85,B 0,C 180,E1 -29702.218,E2 -29702.218} C_VEL
LIN {X 0,Y 73.13,Z 218.19,A -85,B 0,C 180,E1 -29709.106,E2 -29709.106} C_VEL
LIN {X 0,Y 72.144,Z 217.881,A -85,B 0,C 180,E1 -29716.989,E2 -29716.989} C_VEL
LIN {X 0,Y 72.686,Z 218.419,A -85,B 0,C 180,E1 -29727.704,E2 -29727.704} C_VEL
LIN {X 0,Y 74.098,Z 221.626,A -85,B 0,C 180,E1 -29735.124,E2 -29735.124} C_VEL
LIN {X 0,Y 74.936,Z 222.979,A -85,B 0,C 180,E1 -29738.055,E2 -29738.055} C_VEL
LIN {X 0,Y 77.019,Z 226.967,A -85,B 0,C 180,E1 -29743.786,E2 -29743.786} C_VEL
LIN {X 0,Y 79.839,Z 232.461,A -85,B 0,C 180,E1 -29749.557,E2 -29749.557} C_VEL
LIN {X 0,Y 83.082,Z 239.85,A -85,B 0,C 180,E1 -29755.082,E2 -29755.082} C_VEL
LIN {X 0,Y 85.218,Z 245.105,A -85,B 0,C 180,E1 -29758.172,E2 -29758.172} C_VEL
LIN {X 0,Y 85.981,Z 247.328,A -85,B 0,C 180,E1 -29759.243,E2 -29759.243} C_VEL
LIN {X 0,Y 86.476,Z 249.694,A -85,B 0,C 180,E1 -29760.051,E2 -29760.051} C_VEL
LIN {X 0,Y 86.309,Z 253.322,A -85,B 0,C 180,E1 -29760.454,E2 -29760.454} C_VEL
LIN {X 0,Y 85.185,Z 258.052,A -85,B 0,C 180,E1 -29760.197,E2 -29760.197} C_VEL
LIN {X 0,Y 79.823,Z 271.622,A -85,B 0,C 180,E1 -29757.593,E2 -29757.593} C_VEL
LIN {X 0,Y 78.35,Z 276.838,A -85,B 0,C 180,E1 -29757.334,E2 -29757.334} C_VEL
LIN {X 0,Y 78.158,Z 277.9,A -85,B 0,C 180,E1 -29757.426,E2 -29757.426} C_VEL
LIN {X 0,Y 75.203,Z 291.089,A -85,B 0,C 180,E1 -29758.799,E2 -29758.799} C_VEL
LIN {X 0,Y 71.165,Z 303.779,A -85,B 0,C 180,E1 -29760.82,E2 -29760.82} C_VEL
LIN {X 0,Y 66.47,Z 314.931,A -85,B 0,C 180,E1 -29763.301,E2 -29763.301} C_VEL
LIN {X 0,Y 60.649,Z 326.277,A -85,B 0,C 180,E1 -29766.997,E2 -29766.997} C_VEL
LIN {X 0,Y 54.42,Z 336.688,A -85,B 0,C 180,E1 -29772.143,E2 -29772.143} C_VEL
LIN {X 0,Y 47.657,Z 346.594,A -85,B 0,C 180,E1 -29779.758,E2 -29779.758} C_VEL
LIN {X 0,Y 41.646,Z 355.013,A -85,B 0,C 180,E1 -29790.006,E2 -29790.006} C_VEL
LIN {X 0,Y 37.107,Z 361.919,A -85,B 0,C 180,E1 -29803.145,E2 -29803.145} C_VEL
LIN {X 0,Y 34.414,Z 367.546,A -85,B 0,C 180,E1 -29818.943,E2 -29818.943} C_VEL
LIN {X 0,Y 34.263,Z 372.004,A -85,B 0,C 180,E1 -29835.822,E2 -29835.822} C_VEL
LIN {X 0,Y 38.315,Z 376.559,A -85,B 0,C 180,E1 -29856.525,E2 -29856.525} C_VEL
LIN {X 0,Y 45.513,Z 379.423,A -85,B 0,C 180,E1 -29871.122,E2 -29871.122} C_VEL
LIN {X 0,Y 56.289,Z 381.201,A -85,B 0,C 180,E1 -29882.674,E2 -29882.674} C_VEL
LIN {X 0,Y 63.85,Z 381.462,A -85,B 0,C 180,E1 -29887.819,E2 -29887.819} C_VEL
LIN {X 0,Y 71.796,Z 381.147,A -85,B 0,C 180,E1 -29891.778,E2 -29891.778} C_VEL
LIN {X 0,Y 84.754,Z 379.33,A -85,B 0,C 180,E1 -29896.437,E2 -29896.437} C_VEL
LIN {X 0,Y 86.726,Z 378.942,A -85,B 0,C 180,E1 -29897,E2 -29897} C_VEL
LIN {X 0,Y 83.685,Z 379.699,A -85,B 0,C 180,E1 -29898.628,E2 -29898.628} C_VEL
LIN {X 0,Y 75.461,Z 381.249,A -85,B 0,C 180,E1 -29901.346,E2 -29901.346} C_VEL
LIN {X 0,Y 63.14,Z 382.49,A -85,B 0,C 180,E1 -29907.06,E2 -29907.06} C_VEL
LIN {X 0,Y 51.81,Z 382.366,A -85,B 0,C 180,E1 -29915.513,E2 -29915.513} C_VEL
LIN {X 0,Y 46.723,Z 381.777,A -85,B 0,C 180,E1 -29921.22,E2 -29921.22} C_VEL
LIN {X 0,Y 38.863,Z 379.523,A -85,B 0,C 180,E1 -29937.138,E2 -29937.138} C_VEL
LIN {X 0,Y 35.267,Z 375.806,A -85,B 0,C 180,E1 -29958.498,E2 -29958.498} C_VEL
LIN {X 0,Y 35.046,Z 373.271,A -85,B 0,C 180,E1 -29969.993,E2 -29969.993} C_VEL
LIN {X 0,Y 36.01,Z 367.184,A -85,B 0,C 180,E1 -29989.964,E2 -29989.964} C_VEL
LIN {X 0,Y 39.733,Z 360.466,A -85,B 0,C 180,E1 -30005.083,E2 -30005.083} C_VEL
LIN {X 0,Y 45.623,Z 352.083,A -85,B 0,C 180,E1 -30017.023,E2 -30017.023} C_VEL
LIN {X 0,Y 51.689,Z 343.433,A -85,B 0,C 180,E1 -30024.658,E2 -30024.658} C_VEL
LIN {X 0,Y 57.984,Z 333.675,A -85,B 0,C 180,E1 -30030.192,E2 -30030.192} C_VEL
LIN {X 0,Y 64.27,Z 322.315,A -85,B 0,C 180,E1 -30034.434,E2 -30034.434} C_VEL
LIN {X 0,Y 69.553,Z 310.721,A -85,B 0,C 180,E1 -30037.218,E2 -30037.218} C_VEL
LIN {X 0,Y 74.176,Z 297.656,A -85,B 0,C 180,E1 -30039.323,E2 -30039.323} C_VEL
LIN {X 0,Y 77.453,Z 284.884,A -85,B 0,C 180,E1 -30040.621,E2 -30040.621} C_VEL
LIN {X 0,Y 80.03,Z 268.134,A -85,B 0,C 180,E1 -30041.665,E2 -30041.665} C_VEL
LIN {X 0,Y 81.719,Z 254.583,A -85,B 0,C 180,E1 -30042.454,E2 -30042.454} C_VEL
LIN {X 0,Y 79.777,Z 245.264,A -85,B 0,C 180,E1 -30046.505,E2 -30046.505} C_VEL
LIN {X 0,Y 77.497,Z 239.007,A -85,B 0,C 180,E1 -30051.117,E2 -30051.117} C_VEL
LIN {X 0,Y 75.453,Z 234.133,A -85,B 0,C 180,E1 -30055.863,E2 -30055.863} C_VEL
LIN {X 0,Y 73.704,Z 229.905,A -85,B 0,C 180,E1 -30061.178,E2 -30061.178} C_VEL
LIN {X 0,Y 72.915,Z 227.974,A -85,B 0,C 180,E1 -30064.345,E2 -30064.345} C_VEL
LIN {X 0,Y 71.901,Z 225.177,A -85,B 0,C 180,E1 -30069.931,E2 -30069.931} C_VEL
LIN {X 0,Y 71.089,Z 224.885,A -85,B 0,C 180,E1 -30077.249,E2 -30077.249} C_VEL
LIN {X 0,Y 71.462,Z 225.349,A -85,B 0,C 180,E1 -30086.513,E2 -30086.513} C_VEL
LIN {X 0,Y 72.922,Z 228.757,A -85,B 0,C 180,E1 -30094.898,E2 -30094.898} C_VEL
LIN {X 0,Y 74.868,Z 233.024,A -85,B 0,C 180,E1 -30101.506,E2 -30101.506} C_VEL
LIN {X 0,Y 77.388,Z 238.565,A -85,B 0,C 180,E1 -30107.505,E2 -30107.505} C_VEL
LIN {X 0,Y 80.294,Z 245.984,A -85,B 0,C 180,E1 -30113.133,E2 -30113.133} C_VEL
LIN {X 0,Y 81.905,Z 250.677,A -85,B 0,C 180,E1 -30115.881,E2 -30115.881} C_VEL
LIN {X 0,Y 78.35,Z 276.842,A -85,B 0,C 180,E1 -30117.335,E2 -30117.335} C_VEL
LIN {X 0,Y 78.158,Z 277.9,A -85,B 0,C 180,E1 -30117.426,E2 -30117.426} C_VEL
LIN {X 0,Y 77.286,Z 281.727,A -85,B 0,C 180,E1 -30117.586,E2 -30117.586} C_VEL
LIN {X 0,Y 75.285,Z 287.298,A -85,B 0,C 180,E1 -30117.352,E2 -30117.352} C_VEL
LIN {X 0,Y 68.667,Z 300.629,A -85,B 0,C 180,E1 -30116.074,E2 -30116.074} C_VEL
LIN {X 0,Y 65.821,Z 306.891,A -85,B 0,C 180,E1 -30116.594,E2 -30116.594} C_VEL
LIN {X 0,Y 60.174,Z 318.849,A -85,B 0,C 180,E1 -30119.276,E2 -30119.276} C_VEL
LIN {X 0,Y 53.52,Z 330.333,A -85,B 0,C 180,E1 -30123.39,E2 -30123.39} C_VEL
LIN {X 0,Y 46.723,Z 340.32,A -85,B 0,C 180,E1 -30128.989,E2 -30128.989} C_VEL
LIN {X 0,Y 39.816,Z 349.373,A -85,B 0,C 180,E1 -30137.26,E2 -30137.26} C_VEL
LIN {X 0,Y 33.296,Z 357.571,A -85,B 0,C 180,E1 -30150.007,E2 -30150.007} C_VEL
LIN {X 0,Y 28.533,Z 364.399,A -85,B 0,C 180,E1 -30167.945,E2 -30167.945} C_VEL
LIN {X 0,Y 26.945,Z 369.533,A -85,B 0,C 180,E1 -30188.524,E2 -30188.524} C_VEL
LIN {X 0,Y 29.085,Z 374.052,A -85,B 0,C 180,E1 -30211.109,E2 -30211.109} C_VEL
LIN {X 0,Y 35.658,Z 377.81,A -85,B 0,C 180,E1 -30230.261,E2 -30230.261} C_VEL
LIN {X 0,Y 42.301,Z 379.763,A -85,B 0,C 180,E1 -30240.005,E2 -30240.005} C_VEL
LIN {X 0,Y 50.957,Z 381.218,A -85,B 0,C 180,E1 -30247.932,E2 -30247.932} C_VEL
LIN {X 0,Y 60.336,Z 381.835,A -85,B 0,C 180,E1 -30253.475,E2 -30253.475} C_VEL
LIN {X 0,Y 67.87,Z 381.693,A -85,B 0,C 180,E1 -30256.663,E2 -30256.663} C_VEL
LIN {X 0,Y 66.642,Z 381.874,A -85,B 0,C 180,E1 -30258.343,E2 -30258.343} C_VEL
LIN {X 0,Y 53.993,Z 382.193,A -85,B 0,C 180,E1 -30264.325,E2 -30264.325} C_VEL
LIN {X 0,Y 42.384,Z 381.102,A -85,B 0,C 180,E1 -30273.986,E2 -30273.986} C_VEL
LIN {X 0,Y 33.145,Z 378.656,A -85,B 0,C 180,E1 -30290.487,E2 -30290.487} C_VEL
LIN {X 0,Y 29.042,Z 375.821,A -85,B 0,C 180,E1 -30308.707,E2 -30308.707} C_VEL
LIN {X 0,Y 28.207,Z 373.433,A -85,B 0,C 180,E1 -30322.835,E2 -30322.835} C_VEL
LIN {X 0,Y 27.906,Z 370.374,A -85,B 0,C 180,E1 -30337.226,E2 -30337.226} C_VEL
LIN {X 0,Y 30.065,Z 364.609,A -85,B 0,C 180,E1 -30357.865,E2 -30357.865} C_VEL
LIN {X 0,Y 35.227,Z 357.338,A -85,B 0,C 180,E1 -30374.279,E2 -30374.279} C_VEL
LIN {X 0,Y 41.079,Z 349.89,A -85,B 0,C 180,E1 -30384.346,E2 -30384.346} C_VEL
LIN {X 0,Y 47.945,Z 340.914,A -85,B 0,C 180,E1 -30391.574,E2 -30391.574} C_VEL
LIN {X 0,Y 54.739,Z 330.817,A -85,B 0,C 180,E1 -30396.559,E2 -30396.559} C_VEL
LIN {X 0,Y 60.76,Z 320.062,A -85,B 0,C 180,E1 -30400.007,E2 -30400.007} C_VEL
LIN {X 0,Y 66.333,Z 307.99,A -85,B 0,C 180,E1 -30402.457,E2 -30402.457} C_VEL
LIN {X 0,Y 70.771,Z 295.381,A -85,B 0,C 180,E1 -30404.147,E2 -30404.147} C_VEL
LIN {X 0,Y 74.244,Z 281.208,A -85,B 0,C 180,E1 -30405.312,E2 -30405.312} C_VEL
LIN {X 0,Y 77.736,Z 256.547,A -85,B 0,C 180,E1 -30406.62,E2 -30406.62} C_VEL
LIN {X 0,Y 76.558,Z 249.722,A -85,B 0,C 180,E1 -30409.836,E2 -30409.836} C_VEL
LIN {X 0,Y 74.738,Z 244.153,A -85,B 0,C 180,E1 -30414.207,E2 -30414.207} C_VEL
LIN {X 0,Y 73.206,Z 239.872,A -85,B 0,C 180,E1 -30418.602,E2 -30418.602} C_VEL
LIN {X 0,Y 71.821,Z 235.782,A -85,B 0,C 180,E1 -30424.011,E2 -30424.011} C_VEL
LIN {X 0,Y 71.198,Z 234.059,A -85,B 0,C 180,E1 -30427.129,E2 -30427.129} C_VEL
LIN {X 0,Y 70.587,Z 232.055,A -85,B 0,C 180,E1 -30431.483,E2 -30431.483} C_VEL
LIN {X 0,Y 70.146,Z 232.074,A -85,B 0,C 180,E1 -30443.622,E2 -30443.622} C_VEL
LIN {X 0,Y 70.282,Z 232.335,A -85,B 0,C 180,E1 -30445.464,E2 -30445.464} C_VEL
LIN {X 0,Y 71.619,Z 236.005,A -85,B 0,C 180,E1 -30454.326,E2 -30454.326} C_VEL
LIN {X 0,Y 72.995,Z 239.501,A -85,B 0,C 180,E1 -30459.629,E2 -30459.629} C_VEL
LIN {X 0,Y 75.15,Z 245.023,A -85,B 0,C 180,E1 -30465.644,E2 -30465.644} C_VEL
LIN {X 0,Y 77.879,Z 252.979,A -85,B 0,C 180,E1 -30471.613,E2 -30471.613} C_VEL
LIN {X 0,Y 75.343,Z 272.138,A -85,B 0,C 180,E1 -30472.646,E2 -30472.646} C_VEL
LIN {X 0,Y 72.54,Z 286.191,A -85,B 0,C 180,E1 -30473.617,E2 -30473.617} C_VEL
LIN {X 0,Y 68.759,Z 299.125,A -85,B 0,C 180,E1 -30475.263,E2 -30475.263} C_VEL
LIN {X 0,Y 65.821,Z 306.891,A -85,B 0,C 180,E1 -30476.594,E2 -30476.594} C_VEL
LIN {X 0,Y 63.228,Z 312.15,A -85,B 0,C 180,E1 -30477.202,E2 -30477.202} C_VEL
LIN {X 0,Y 57.512,Z 320.259,A -85,B 0,C 180,E1 -30476.893,E2 -30476.893} C_VEL
LIN {X 0,Y 51.186,Z 327.968,A -85,B 0,C 180,E1 -30476.761,E2 -30476.761} C_VEL
LIN {X 0,Y 47.642,Z 332.61,A -85,B 0,C 180,E1 -30478.008,E2 -30478.008} C_VEL
LIN {X 0,Y 40.327,Z 342.309,A -85,B 0,C 180,E1 -30483.566,E2 -30483.566} C_VEL
LIN {X 0,Y 33.329,Z 350.508,A -85,B 0,C 180,E1 -30491.568,E2 -30491.568} C_VEL
LIN {X 0,Y 25.755,Z 358.936,A -85,B 0,C 180,E1 -30506.968,E2 -30506.968} C_VEL
LIN {X 0,Y 20.902,Z 365.347,A -85,B 0,C 180,E1 -30529.66,E2 -30529.66} C_VEL
LIN {X 0,Y 20.004,Z 369.919,A -85,B 0,C 180,E1 -30555.375,E2 -30555.375} C_VEL
LIN {X 0,Y 23.922,Z 374.386,A -85,B 0,C 180,E1 -30582.925,E2 -30582.925} C_VEL
LIN {X 0,Y 31.295,Z 377.729,A -85,B 0,C 180,E1 -30600.007,E2 -30600.007} C_VEL
LIN {X 0,Y 43.174,Z 380.67,A -85,B 0,C 180,E1 -30612.37,E2 -30612.37} C_VEL
LIN {X 0,Y 49.799,Z 381.567,A -85,B 0,C 180,E1 -30616.399,E2 -30616.399} C_VEL
LIN {X 0,Y 45.07,Z 381.237,A -85,B 0,C 180,E1 -30620.659,E2 -30620.659} C_VEL
LIN {X 0,Y 38.867,Z 380.413,A -85,B 0,C 180,E1 -30625.282,E2 -30625.282} C_VEL
LIN {X 0,Y 28.053,Z 377.728,A -85,B 0,C 180,E1 -30641.26,E2 -30641.26} C_VEL
LIN {X 0,Y 21.702,Z 373.515,A -85,B 0,C 180,E1 -30671.093,E2 -30671.093} C_VEL
LIN {X 0,Y 21.29,Z 372.208,A -85,B 0,C 180,E1 -30680.489,E2 -30680.489} C_VEL
LIN {X 0,Y 20.929,Z 368.956,A -85,B 0,C 180,E1 -30699.655,E2 -30699.655} C_VEL
LIN {X 0,Y 24.013,Z 362.924,A -85,B 0,C 180,E1 -30725.816,E2 -30725.816} C_VEL
LIN {X 0,Y 30.568,Z 355.372,A -85,B 0,C 180,E1 -30743.569,E2 -30743.569} C_VEL
LIN {X 0,Y 38.883,Z 345.814,A -85,B 0,C 180,E1 -30754.641,E2 -30754.641} C_VEL
LIN {X 0,Y 46.581,Z 336.019,A -85,B 0,C 180,E1 -30760.543,E2 -30760.543} C_VEL
LIN {X 0,Y 53.363,Z 325.777,A -85,B 0,C 180,E1 -30764.235,E2 -30764.235} C_VEL
LIN {X 0,Y 59.56,Z 314.392,A -85,B 0,C 180,E1 -30766.761,E2 -30766.761} C_VEL
LIN {X 0,Y 64.561,Z 302.842,A -85,B 0,C 180,E1 -30768.425,E2 -30768.425} C_VEL
LIN {X 0,Y 68.734,Z 289.843,A -85,B 0,C 180,E1 -30769.707,E2 -30769.707} C_VEL
LIN {X 0,Y 71.555,Z 276.722,A -85,B 0,C 180,E1 -30770.462,E2 -30770.462} C_VEL
LIN {X 0,Y 74.147,Z 258.176,A -85,B 0,C 180,E1 -30771.361,E2 -30771.361} C_VEL
LIN {X 0,Y 73.452,Z 253.77,A -85,B 0,C 180,E1 -30773.704,E2 -30773.704} C_VEL
LIN {X 0,Y 71.743,Z 247.527,A -85,B 0,C 180,E1 -30779.184,E2 -30779.184} C_VEL
LIN {X 0,Y 70.193,Z 242.071,A -85,B 0,C 180,E1 -30786.301,E2 -30786.301} C_VEL
LIN {X 0,Y 69.358,Z 239.039,A -85,B 0,C 180,E1 -30792.687,E2 -30792.687} C_VEL
LIN {X 0,Y 69.117,Z 239.14,A -85,B 0,C 180,E1 -30803.996,E2 -30803.996} C_VEL
LIN {X 0,Y 70.073,Z 242.58,A -85,B 0,C 180,E1 -30812.498,E2 -30812.498} C_VEL
LIN {X 0,Y 71.329,Z 246.304,A -85,B 0,C 180,E1 -30818.133,E2 -30818.133} C_VEL
LIN {X 0,Y 72.876,Z 251.316,A -85,B 0,C 180,E1 -30823.391,E2 -30823.391} C_VEL
LIN {X 0,Y 74.188,Z 255.722,A -85,B 0,C 180,E1 -30826.965,E2 -30826.965} C_VEL
LIN {X 0,Y 73.109,Z 264.231,A -85,B 0,C 180,E1 -30827.502,E2 -30827.502} C_VEL
LIN {X 0,Y 70.297,Z 281.021,A -85,B 0,C 180,E1 -30828.238,E2 -30828.238} C_VEL
LIN {X 0,Y 67.221,Z 292.945,A -85,B 0,C 180,E1 -30829.305,E2 -30829.305} C_VEL
LIN {X 0,Y 62.758,Z 305.273,A -85,B 0,C 180,E1 -30830.912,E2 -30830.912} C_VEL
LIN {X 0,Y 57.053,Z 317.245,A -85,B 0,C 180,E1 -30833.098,E2 -30833.098} C_VEL
LIN {X 0,Y 50.591,Z 328.233,A -85,B 0,C 180,E1 -30836.249,E2 -30836.249} C_VEL
LIN {X 0,Y 47.642,Z 332.61,A -85,B 0,C 180,E1 -30838.008,E2 -30838.008} C_VEL
LIN {X 0,Y 44.007,Z 337.12,A -85,B 0,C 180,E1 -30839.564,E2 -30839.564} C_VEL
LIN {X 0,Y 36.841,Z 343.935,A -85,B 0,C 180,E1 -30840.619,E2 -30840.619} C_VEL
LIN {X 0,Y 29.198,Z 350.244,A -85,B 0,C 180,E1 -30842.505,E2 -30842.505} C_VEL
LIN {X 0,Y 24.937,Z 353.926,A -85,B 0,C 180,E1 -30846.53,E2 -30846.53} C_VEL
LIN {X 0,Y 17.492,Z 361,A -85,B 0,C 180,E1 -30864.248,E2 -30864.248} C_VEL
LIN {X 0,Y 12.867,Z 367.364,A -85,B 0,C 180,E1 -30903.13,E2 -30903.13} C_VEL
LIN {X 0,Y 17.36,Z 373.244,A -85,B 0,C 180,E1 -30951.515,E2 -30951.515} C_VEL
LIN {X 0,Y 28.879,Z 377.874,A -85,B 0,C 180,E1 -30973.195,E2 -30973.195} C_VEL
LIN {X 0,Y 31.895,Z 378.738,A -85,B 0,C 180,E1 -30975.944,E2 -30975.944} C_VEL
LIN {X 0,Y 30.009,Z 378.371,A -85,B 0,C 180,E1 -30980.462,E2 -30980.462} C_VEL
LIN {X 0,Y 18.797,Z 374.699,A -85,B 0,C 180,E1 -31001.582,E2 -31001.582} C_VEL
LIN {X 0,Y 14.439,Z 370.892,A -85,B 0,C 180,E1 -31035.897,E2 -31035.897} C_VEL
LIN {X 0,Y 14.014,Z 367.521,A -85,B 0,C 180,E1 -31064.505,E2 -31064.505} C_VEL
LIN {X 0,Y 18.727,Z 361.203,A -85,B 0,C 180,E1 -31098.62,E2 -31098.62} C_VEL
LIN {X 0,Y 26.974,Z 353.264,A -85,B 0,C 180,E1 -31115.749,E2 -31115.749} C_VEL
LIN {X 0,Y 34.798,Z 345.123,A -85,B 0,C 180,E1 -31123.58,E2 -31123.58} C_VEL
LIN {X 0,Y 43.05,Z 335.25,A -85,B 0,C 180,E1 -31128.354,E2 -31128.354} C_VEL
LIN {X 0,Y 50.459,Z 324.438,A -85,B 0,C 180,E1 -31131.279,E2 -31131.279} C_VEL
LIN {X 0,Y 56.634,Z 313.365,A -85,B 0,C 180,E1 -31133.071,E2 -31133.071} C_VEL
LIN {X 0,Y 62.228,Z 300.502,A -85,B 0,C 180,E1 -31134.388,E2 -31134.388} C_VEL
LIN {X 0,Y 66.438,Z 286.863,A -85,B 0,C 180,E1 -31135.304,E2 -31135.304} C_VEL
LIN {X 0,Y 69.069,Z 273.834,A -85,B 0,C 180,E1 -31135.825,E2 -31135.825} C_VEL
LIN {X 0,Y 70.984,Z 260.046,A -85,B 0,C 180,E1 -31136.452,E2 -31136.452} C_VEL
LIN {X 0,Y 70.511,Z 257.012,A -85,B 0,C 180,E1 -31138.549,E2 -31138.549} C_VEL
LIN {X 0,Y 69.396,Z 251.901,A -85,B 0,C 180,E1 -31143.811,E2 -31143.811} C_VEL
LIN {X 0,Y 68.526,Z 247.686,A -85,B 0,C 180,E1 -31149.768,E2 -31149.768} C_VEL
LIN {X 0,Y 68.192,Z 246.036,A -85,B 0,C 180,E1 -31153.611,E2 -31153.611} C_VEL
LIN {X 0,Y 67.995,Z 246.222,A -85,B 0,C 180,E1 -31163.186,E2 -31163.186} C_VEL
LIN {X 0,Y 68.628,Z 249.281,A -85,B 0,C 180,E1 -31170.796,E2 -31170.796} C_VEL
LIN {X 0,Y 69.516,Z 252.523,A -85,B 0,C 180,E1 -31175.721,E2 -31175.721} C_VEL
LIN {X 0,Y 70.771,Z 257.687,A -85,B 0,C 180,E1 -31181.139,E2 -31181.139} C_VEL
LIN {X 0,Y 71.032,Z 258.919,A -85,B 0,C 180,E1 -31182.134,E2 -31182.134} C_VEL
LIN {X 0,Y 67.627,Z 279.926,A -85,B 0,C 180,E1 -31182.794,E2 -31182.794} C_VEL
LIN {X 0,Y 64.462,Z 292.22,A -85,B 0,C 180,E1 -31183.639,E2 -31183.639} C_VEL
LIN {X 0,Y 59.58,Z 305.448,A -85,B 0,C 180,E1 -31184.953,E2 -31184.953} C_VEL
LIN {X 0,Y 53.69,Z 317.381,A -85,B 0,C 180,E1 -31186.595,E2 -31186.595} C_VEL
LIN {X 0,Y 46.9,Z 328.438,A -85,B 0,C 180,E1 -31189.064,E2 -31189.064} C_VEL
LIN {X 0,Y 39.295,Z 338.582,A -85,B 0,C 180,E1 -31192.877,E2 -31192.877} C_VEL
LIN {X 0,Y 31.576,Z 347.299,A -85,B 0,C 180,E1 -31198.632,E2 -31198.632} C_VEL
LIN {X 0,Y 24.937,Z 353.926,A -85,B 0,C 180,E1 -31206.53,E2 -31206.53} C_VEL
LIN {X 0,Y 20.714,Z 357.425,A -85,B 0,C 180,E1 -31212.158,E2 -31212.158} C_VEL
LIN {X 0,Y 12.831,Z 362.51,A -85,B 0,C 180,E1 -31223.555,E2 -31223.555} C_VEL
LIN {X 0,Y 6.418,Z 367.004,A -85,B 0,C 180,E1 -31263.898,E2 -31263.898} C_VEL
LIN {X 0,Y 7.51,Z 369.543,A -85,B 0,C 180,E1 -31308.778,E2 -31308.778} C_VEL
LIN {X 0,Y 14.622,Z 373.275,A -85,B 0,C 180,E1 -31335.938,E2 -31335.938} C_VEL
LIN {X 0,Y 15.077,Z 373.526,A -85,B 0,C 180,E1 -31341.162,E2 -31341.162} C_VEL
LIN {X 0,Y 7.839,Z 369.525,A -85,B 0,C 180,E1 -31383.335,E2 -31383.335} C_VEL
LIN {X 0,Y 9.366,Z 363.91,A -85,B 0,C 180,E1 -31458.584,E2 -31458.584} C_VEL
LIN {X 0,Y 18.234,Z 356.754,A -85,B 0,C 180,E1 -31484.439,E2 -31484.439} C_VEL
LIN {X 0,Y 26.618,Z 349.468,A -85,B 0,C 180,E1 -31491.883,E2 -31491.883} C_VEL
LIN {X 0,Y 35.23,Z 340.641,A -85,B 0,C 180,E1 -31495.805,E2 -31495.805} C_VEL
LIN {X 0,Y 43.071,Z 330.996,A -85,B 0,C 180,E1 -31497.93,E2 -31497.93} C_VEL
LIN {X 0,Y 50.562,Z 319.533,A -85,B 0,C 180,E1 -31499.42,E2 -31499.42} C_VEL
LIN {X 0,Y 57.099,Z 306.764,A -85,B 0,C 180,E1 -31500.322,E2 -31500.322} C_VEL
LIN {X 0,Y 61.925,Z 294.102,A -85,B 0,C 180,E1 -31500.925,E2 -31500.925} C_VEL
LIN {X 0,Y 65.463,Z 280.851,A -85,B 0,C 180,E1 -31501.273,E2 -31501.273} C_VEL
LIN {X 0,Y 68.377,Z 262.519,A -85,B 0,C 180,E1 -31501.853,E2 -31501.853} C_VEL
LIN {X 0,Y 67.646,Z 257.782,A -85,B 0,C 180,E1 -31506.819,E2 -31506.819} C_VEL
LIN {X 0,Y 67.136,Z 253.972,A -85,B 0,C 180,E1 -31512.469,E2 -31512.469} C_VEL
LIN {X 0,Y 67.038,Z 253.068,A -85,B 0,C 180,E1 -31514.568,E2 -31514.568} C_VEL
LIN {X 0,Y 66.902,Z 253.05,A -85,B 0,C 180,E1 -31521.771,E2 -31521.771} C_VEL
LIN {X 0,Y 67.199,Z 255.722,A -85,B 0,C 180,E1 -31528.538,E2 -31528.538} C_VEL
LIN {X 0,Y 67.819,Z 259.024,A -85,B 0,C 180,E1 -31533.491,E2 -31533.491} C_VEL
LIN {X 0,Y 68.358,Z 262.053,A -85,B 0,C 180,E1 -31536.67,E2 -31536.67} C_VEL
LIN {X 0,Y 65.169,Z 280.87,A -85,B 0,C 180,E1 -31537.042,E2 -31537.042} C_VEL
LIN {X 0,Y 61.677,Z 293.697,A -85,B 0,C 180,E1 -31537.644,E2 -31537.644} C_VEL
LIN {X 0,Y 57.102,Z 305.564,A -85,B 0,C 180,E1 -31538.408,E2 -31538.408} C_VEL
LIN {X 0,Y 51.127,Z 317.38,A -85,B 0,C 180,E1 -31539.362,E2 -31539.362} C_VEL
LIN {X 0,Y 43.607,Z 329.162,A -85,B 0,C 180,E1 -31540.955,E2 -31540.955} C_VEL
LIN {X 0,Y 35.124,Z 339.784,A -85,B 0,C 180,E1 -31543.514,E2 -31543.514} C_VEL
LIN {X 0,Y 26.019,Z 349.169,A -85,B 0,C 180,E1 -31547.872,E2 -31547.872} C_VEL
LIN {X 0,Y 16.848,Z 357.091,A -85,B 0,C 180,E1 -31556.516,E2 -31556.516} C_VEL
LIN {X 0,Y 8.837,Z 363.287,A -85,B 0,C 180,E1 -31578.559,E2 -31578.559} C_VEL
LIN {X 0,Y 7.51,Z 369.543,A -85,B 0,C 180,E1 -31668.778,E2 -31668.778} C_VEL
LIN {X 0,Y 6.507,Z 369.239,A -85,B 0,C 180,E1 -31671.419,E2 -31671.419} C_VEL
LIN {X 0,Y 5.437,Z 368.722,A -85,B 0,C 180,E1 -31669.582,E2 -31669.582} C_VEL
LIN {X 0,Y 2.887,Z 365.228,A -85,B 0,C 180,E1 -31573.448,E2 -31573.448} C_VEL
LIN {X 0,Y 10.935,Z 359.539,A -85,B 0,C 180,E1 -31535.294,E2 -31535.294} C_VEL
LIN {X 0,Y 15.76,Z 355.95,A -85,B 0,C 180,E1 -31532.656,E2 -31532.656} C_VEL
LIN {X 0,Y 20.447,Z 352.14,A -85,B 0,C 180,E1 -31532.118,E2 -31532.118} C_VEL
LIN {X 0,Y 30.087,Z 343.141,A -85,B 0,C 180,E1 -31532.152,E2 -31532.152} C_VEL
LIN {X 0,Y 38.998,Z 332.866,A -85,B 0,C 180,E1 -31531.839,E2 -31531.839} C_VEL
LIN {X 0,Y 47.421,Z 320.698,A -85,B 0,C 180,E1 -31531.56,E2 -31531.56} C_VEL
LIN {X 0,Y 53.9,Z 308.787,A -85,B 0,C 180,E1 -31531.432,E2 -31531.432} C_VEL
LIN {X 0,Y 59.015,Z 296.426,A -85,B 0,C 180,E1 -31531.202,E2 -31531.202} C_VEL
LIN {X 0,Y 62.964,Z 283.21,A -85,B 0,C 180,E1 -31530.915,E2 -31530.915} C_VEL
LIN {X 0,Y 65.73,Z 268.404,A -85,B 0,C 180,E1 -31530.873,E2 -31530.873} C_VEL
LIN {X 0,Y 66.187,Z 265.197,A -85,B 0,C 180,E1 -31530.727,E2 -31530.727} C_VEL
LIN {X 0,Y 65.865,Z 261.787,A -85,B 0,C 180,E1 -31525.587,E2 -31525.587} C_VEL
LIN {X 0,Y 65.814,Z 260.038,A -85,B 0,C 180,E1 -31520.176,E2 -31520.176} C_VEL
LIN {X 0,Y 65.908,Z 260.234,A -85,B 0,C 180,E1 -31515.226,E2 -31515.226} C_VEL
LIN {X 0,Y 65.988,Z 262.74,A -85,B 0,C 180,E1 -31511.248,E2 -31511.248} C_VEL
LIN {X 0,Y 66.241,Z 265.684,A -85,B 0,C 180,E1 -31507.626,E2 -31507.626} C_VEL
LIN {X 0,Y 63.337,Z 282.517,A -85,B 0,C 180,E1 -31507.404,E2 -31507.404} C_VEL
LIN {X 0,Y 59.714,Z 295.31,A -85,B 0,C 180,E1 -31507.38,E2 -31507.38} C_VEL
LIN {X 0,Y 55.05,Z 307.04,A -85,B 0,C 180,E1 -31507.331,E2 -31507.331} C_VEL
LIN {X 0,Y 48.713,Z 319.207,A -85,B 0,C 180,E1 -31507.346,E2 -31507.346} C_VEL
LIN {X 0,Y 41.617,Z 330.005,A -85,B 0,C 180,E1 -31507.236,E2 -31507.236} C_VEL
LIN {X 0,Y 33.646,Z 339.762,A -85,B 0,C 180,E1 -31507.217,E2 -31507.217} C_VEL
LIN {X 0,Y 24.785,Z 348.669,A -85,B 0,C 180,E1 -31507.124,E2 -31507.124} C_VEL
LIN {X 0,Y 14.161,Z 357.361,A -85,B 0,C 180,E1 -31507.107,E2 -31507.107} C_VEL
LIN {X 0,Y 7.074,Z 362.156,A -85,B 0,C 180,E1 -31506.826,E2 -31506.826} C_VEL
LIN {X 0,Y 5.512,Z 362.994,A -85,B 0,C 180,E1 -31524.79,E2 -31524.79} C_VEL
LIN {X 0,Y 15.027,Z 356.477,A -85,B 0,C 180,E1 -31531.773,E2 -31531.773} C_VEL
LIN {X 0,Y 20.447,Z 352.14,A -85,B 0,C 180,E1 -31532.118,E2 -31532.118} C_VEL
LIN {X 0,Y 23.478,Z 349.456,A -85,B 0,C 180,E1 -31531.206,E2 -31531.206} C_VEL
LIN {X 0,Y 26.332,Z 346.694,A -85,B 0,C 180,E1 -31529.108,E2 -31529.108} C_VEL
LIN {X 0,Y 31.671,Z 340.96,A -85,B 0,C 180,E1 -31523.849,E2 -31523.849} C_VEL
LIN {X 0,Y 36.826,Z 334.902,A -85,B 0,C 180,E1 -31519.228,E2 -31519.228} C_VEL
LIN {X 0,Y 40.556,Z 330.039,A -85,B 0,C 180,E1 -31517.181,E2 -31517.181} C_VEL
LIN {X 0,Y 41.757,Z 328.339,A -85,B 0,C 180,E1 -31516.86,E2 -31516.86} C_VEL
LIN {X 0,Y 49.222,Z 316.471,A -85,B 0,C 180,E1 -31515.484,E2 -31515.484} C_VEL
LIN {X 0,Y 54.988,Z 304.79,A -85,B 0,C 180,E1 -31514.594,E2 -31514.594} C_VEL
LIN {X 0,Y 59.773,Z 291.771,A -85,B 0,C 180,E1 -31514.074,E2 -31514.074} C_VEL
LIN {X 0,Y 63.112,Z 278.732,A -85,B 0,C 180,E1 -31513.765,E2 -31513.765} C_VEL
LIN {X 0,Y 64.693,Z 269.118,A -85,B 0,C 180,E1 -31513.861,E2 -31513.861} C_VEL
LIN {X 0,Y 64.789,Z 267.012,A -85,B 0,C 180,E1 -31517.045,E2 -31517.045} C_VEL
LIN {X 0,Y 64.729,Z 267.286,A -85,B 0,C 180,E1 -31520.245,E2 -31520.245} C_VEL
LIN {X 0,Y 64.676,Z 269.024,A -85,B 0,C 180,E1 -31524.569,E2 -31524.569} C_VEL
LIN {X 0,Y 61.965,Z 283.581,A -85,B 0,C 180,E1 -31524.447,E2 -31524.447} C_VEL
LIN {X 0,Y 57.929,Z 297.002,A -85,B 0,C 180,E1 -31524.298,E2 -31524.298} C_VEL
LIN {X 0,Y 53.055,Z 308.804,A -85,B 0,C 180,E1 -31523.863,E2 -31523.863} C_VEL
LIN {X 0,Y 46.647,Z 320.761,A -85,B 0,C 180,E1 -31522.936,E2 -31522.936} C_VEL
LIN {X 0,Y 38.561,Z 332.611,A -85,B 0,C 180,E1 -31521.372,E2 -31521.372} C_VEL
LIN {X 0,Y 35.612,Z 336.324,A -85,B 0,C 180,E1 -31520.581,E2 -31520.581} C_VEL
LIN {X 0,Y 36.965,Z 334.721,A -85,B 0,C 180,E1 -31518.099,E2 -31518.099} C_VEL
LIN {X 0,Y 41.757,Z 328.339,A -85,B 0,C 180,E1 -31516.86,E2 -31516.86} C_VEL
LIN {X 0,Y 45.368,Z 329.483,A -85,B 0,C 180,E1 -31516.243,E2 -31516.243} C_VEL
LIN {X 0,Y 45.368,Z 600,A -85,B 0,C 180,E1 -31516.243,E2 -31516.243} C_VEL
LIN {X 0,Y 45.368,Z 600,A -85,B 0,C 180,E1 -31516.243,E2 -31516.243}

QRS_NEXT_CUT()

QRS_NEXT()
QRS_HOME()

END
